// TwinCAT 3 PLC project Field_IO
// ProgramVersion: 3.1.4023.0
// libraries:
//   Tc2_Standard, * (Beckhoff Automation GmbH)
//   Tc2_System, * (Beckhoff Automation GmbH)
//   Tc3_Module, * (Beckhoff Automation GmbH)
// project tree:
//   / PlcTask.TcTTO
//   POUs/ Flasher.TcPOU, HB_M2S.TcPOU, MAIN.TcPOU, HB_S2M.TcPOU
// real-time tasks:
//   TASK IO: cycle T#1ms, priority 1, ADS port 301
//   TASK EIP_Sync_Task: cycle T#2ms, priority 2, ADS port 302
//   TASK PlcTask: cycle T#3ms, priority 3, ADS port 350
// I/O:
//   DEVICE Field_Network (TC3 EIP Adapter), AmsNetId 0.0.0.0.3.1
//     BFIO (TC EtherNet/IP Slave)
//     BSIO (TC EtherNet/IP Slave)
//     Movi_1 (TC EtherNet/IP Slave)
//     Movi_2 (TC EtherNet/IP Slave)
//   DEVICE Device 13 (NOV-DP-RAM)
//   DEVICE SLOT-00 BACKPLANE (EtherCAT), AmsNetId 0.0.0.0.2.1
//     PWR-Supply (EK1200) [EK1200-5000 EtherCAT Power supply (2A E-Bus)]
//       Safety-Ctrl (EL6910) [EL6910, TwinSAFE PLC]
//       License (EL6070-0033) [EL6070-0033 1Ch. Licence key terminal, individual licences]
//       LAS_0600_Slot-01 (EL1018) [EL1018 8Ch. Dig. Input 24V, 10µs]
//       LAS_0600_Slot-02 (EL1018) [EL1018 8Ch. Dig. Input 24V, 10µs]
//       LAS_0600_Slot-03 (EL1018) [EL1018 8Ch. Dig. Input 24V, 10µs]
//       LAS_0600_Slot-04 (EL1904) [EL1904, 4 Ch. Safety Input 24V, TwinSAFE]
//         modules: Module 1 (FSOES)
//       LAS_0600_Slot-05 (EL2008) [EL2008 8Ch. Dig. Output 24V, 0.5A]
//       ECAT-Extension (EK1110) [EK1110 EtherCAT extension]
//     MCP-IOLINK (EP6224-2022) [EP6224-2022 (IO Link Master)]
//       modules: Module 1 (DeviceState Inputs Device), Module 2 (DeviceState Inputs), Module 3 (empty), Module 4 (IO-Link Slave), Module 5 (empty), Module 6 (empty)
//   DEVICE SLOT-01-X600-X601 (EtherCAT) (disabled), AmsNetId 0.0.0.0.4.1
//   DEVICE SLOT-02-X600-X601 (EtherCAT), AmsNetId 0.0.0.0.5.1
//   DEVICE SLOT-03-X600-X601 (EtherCAT), AmsNetId 0.0.0.0.7.1
//     BSIO_LLUB-0635_1 (EP1957-0022) [EP1957, 8Ch. Safety Input 24V, 4Ch. Safety Output 24V, 0.5A, TwinSAFE]
//       modules: Module 1 (FSOE), Module 2 (FSOUT), Module 3 (DEVICEIO), Module 4 (FSLOGIC)
//     BFIO_LLUB-0635_1 (EP2338-0002) [EP2338-0002 8 Ch. Dig. Input/Output 24V, 0,5A, M12]
//     BSIO_LLUB-0636_1 (EP1957-0022) [EP1957, 8Ch. Safety Input 24V, 4Ch. Safety Output 24V, 0.5A, TwinSAFE]
//       modules: Module 1 (FSOE), Module 2 (FSOUT), Module 3 (DEVICEIO), Module 4 (FSLOGIC)
//     BFIO_LLUB-0636_1(EP2338-0002) [EP2338-0002 8 Ch. Dig. Input/Output 24V, 0,5A, M12]
//     MOVI_LLUB-0637 (MOVIMOT+MFE72A) [MOVIMOT+MFE72A]
//     LLU-0200 Coupler (EK1100) [EK1100 EtherCAT Coupler (2A E-Bus)]
//       LLU_0200_Slot-01 (EL1018) [EL1018 8Ch. Dig. Input 24V, 10µs]
//       LLU_0200_Slot-02(EL1018) [EL1018 8Ch. Dig. Input 24V, 10µs]
//       LLU_0200_Slot-03 (EL1018) [EL1018 8Ch. Dig. Input 24V, 10µs]
//       LLU_0200_Slot-04 (EL1904) [EL1904, 4 Ch. Safety Input 24V, TwinSAFE]
//         modules: Module 1 (FSOES)
//       LLU_0200_Slot-05 (EL2008) [EL2008 8Ch. Dig. Output 24V, 0.5A]
//       Slot-06 (EK1110) [EK1110 EtherCAT extension]
//     MOVI_LLUB-0241 (MOVIMOT+MFE72A) [MOVIMOT+MFE72A]
//     MOVI_LLUB-0251 (MOVIMOT+MFE72A) [MOVIMOT+MFE72A]
//     BSIO_LLUB-0639_1  (EP1957-0022) [EP1957, 8Ch. Safety Input 24V, 4Ch. Safety Output 24V, 0.5A, TwinSAFE]
//       modules: Module 1 (FSOE), Module 2 (FSOUT), Module 3 (DEVICEIO), Module 4 (FSLOGIC)
//     IOLINK_LLUB-0639_1 (EP6224-2022) [EP6224-2022 (IO Link Master)]
//       modules: Module 1 (DeviceState Inputs Device), Module 2 (DeviceState Inputs), Module 3 (empty), Module 4 (IO-Link Slave), Module 5 (empty), Module 6 (empty)
//     MOVI_LLUB-0639 (MOVITRAC+FSE24B) [MOVITRAC+FSE24B]
//     BSIO_LLUB-0639_2 (EP1957-0022) [EP1957, 8Ch. Safety Input 24V, 4Ch. Safety Output 24V, 0.5A, TwinSAFE]
//       modules: Module 1 (FSOE), Module 2 (FSOUT), Module 3 (DEVICEIO), Module 4 (FSLOGIC)
//     BSIO_LLUB-0639_2 (EP2338-0002) [EP2338-0002 8 Ch. Dig. Input/Output 24V, 0,5A, M12]
//     BSIO_LLUB-0639_3 (EP1957-0022) [EP1957, 8Ch. Safety Input 24V, 4Ch. Safety Output 24V, 0.5A, TwinSAFE]
//       modules: Module 1 (FSOE), Module 2 (FSOUT), Module 3 (DEVICEIO), Module 4 (FSLOGIC)
//     MOVI_LLUB-0638 (MOVIMOT+MFE72A) [MOVIMOT+MFE72A]
//     MOVI_LLUB-0636 (MOVITRAC+FSE24B) [MOVITRAC+FSE24B]
//     MOVI_LLUB-0635 (MOVITRAC+FSE24B) [MOVITRAC+FSE24B]
//   DEVICE SLOT-04-X600-X601 (EtherCAT), AmsNetId 0.0.0.0.8.1
//     BFIO-LASB-0622_1 (EP2338-0002) [EP2338-0002 8 Ch. Dig. Input/Output 24V, 0,5A, M12]
//     MOVI-LASB-0625 (MOVIMOT+MFE72A) [MOVIMOT+MFE72A]
//     MOVI-LASR-0624 (MOVIMOT+MFE72A) [MOVIMOT+MFE72A]
//     BFIO-LASB-0620_1 (EP2338-0002) [EP2338-0002 8 Ch. Dig. Input/Output 24V, 0,5A, M12]
//     BSIO-LASB-0622_1 (EP1957-0022) [EP1957, 8Ch. Safety Input 24V, 4Ch. Safety Output 24V, 0.5A, TwinSAFE]
//       modules: Module 1 (FSOE), Module 2 (FSOUT), Module 3 (DEVICEIO), Module 4 (FSLOGIC)
//     MOVI-LASB-0626 (MOVIMOT+MFE72A) [MOVIMOT+MFE72A]
//     MOVI-LASB-0629 (MOVIMOT+MFE72A) [MOVIMOT+MFE72A]
//     MOVI-LASB-0628 (MOVIMOT+MFE72A) [MOVIMOT+MFE72A]
//     MOVI-LASB-0627 (MOVIMOT+MFE72A) [MOVIMOT+MFE72A]
//     BSIO-LASB-0623_1 (EP1957-0022) [EP1957, 8Ch. Safety Input 24V, 4Ch. Safety Output 24V, 0.5A, TwinSAFE]
//       modules: Module 1 (FSOE), Module 2 (FSOUT), Module 3 (DEVICEIO), Module 4 (FSLOGIC)
//     MOVI-LASR-0632 (MOVIMOT+MFE72A) [MOVIMOT+MFE72A]
//     MOVI-LASR-0631 (MOVIMOT+MFE72A) [MOVIMOT+MFE72A]
//     MOVI-LASR-0630 (MOVIMOT+MFE72A) [MOVIMOT+MFE72A]
//     MOVI-LASB-0623 (MOVIMOT+MFE72A) [MOVIMOT+MFE72A]
//     MOVI-LASB-0633 (MOVIMOT+MFE72A) [MOVIMOT+MFE72A]
//     MOVI-LASB-0634 (MOVIMOT+MFE72A) [MOVIMOT+MFE72A]
//     BSIO-LASB-0633_1 (EP1957-0022) [EP1957, 8Ch. Safety Input 24V, 4Ch. Safety Output 24V, 0.5A, TwinSAFE]
//       modules: Module 1 (FSOE), Module 2 (FSOUT), Module 3 (DEVICEIO), Module 4 (FSLOGIC)
//     BSIO-LASB-0629_1 (EP1957-0022) [EP1957, 8Ch. Safety Input 24V, 4Ch. Safety Output 24V, 0.5A, TwinSAFE]
//       modules: Module 1 (FSOE), Module 2 (FSOUT), Module 3 (DEVICEIO), Module 4 (FSLOGIC)
//     BSIO-LASB-0625_1 (EP1957-0022) [EP1957, 8Ch. Safety Input 24V, 4Ch. Safety Output 24V, 0.5A, TwinSAFE]
//       modules: Module 1 (FSOE), Module 2 (FSOUT), Module 3 (DEVICEIO), Module 4 (FSLOGIC)
// variable links:
//   Field_Network (TC3 EIP Adapter) <-> SLOT-00 BACKPLANE (EtherCAT)/MCP-IOLINK (EP6224-2022)
//     BFIO (TC EtherNet/IP Slave)/Assembly 1 (Input/Output)/Inputs/M2S_BFIO_301 <-> Module 4 (IO-Link Slave)/IO-Link Port2_out/Port2: process data[1]
//   Field_Network (TC3 EIP Adapter) <-> SLOT-00 BACKPLANE (EtherCAT)/PWR-Supply (EK1200)/LAS_0600_Slot-01 (EL1018)
//     BFIO (TC EtherNet/IP Slave)/Assembly 1 (Input/Output)/Outputs/S2M_BFIO_1 @bit 4 <-> Channel 5/Input
//   Field_Network (TC3 EIP Adapter) <-> SLOT-00 BACKPLANE (EtherCAT)/PWR-Supply (EK1200)/LAS_0600_Slot-02 (EL1018)
//     BFIO (TC EtherNet/IP Slave)/Assembly 1 (Input/Output)/Outputs/S2M_BFIO_2 @bit 5 <-> Channel 6/Input
//   Field_Network (TC3 EIP Adapter) <-> SLOT-00 BACKPLANE (EtherCAT)/PWR-Supply (EK1200)/LAS_0600_Slot-03 (EL1018)
//     BFIO (TC EtherNet/IP Slave)/Assembly 1 (Input/Output)/Outputs/S2M_BFIO_3 <-> Channel 1/Input
//     BFIO (TC EtherNet/IP Slave)/Assembly 1 (Input/Output)/Outputs/S2M_BFIO_3 @bit {1..7} <-> Channel {2..8}/Input  (7 links)
//   Field_Network (TC3 EIP Adapter) <-> SLOT-00 BACKPLANE (EtherCAT)/PWR-Supply (EK1200)/LAS_0600_Slot-04 (EL1904)
//     BSIO (TC EtherNet/IP Slave)/Assembly 3 (Input/Output)/Outputs/S2M_BSIO__11 @bit 3 <-> Module 1 (FSOES)/TxPDO/FSOE/InputChannel4
//   Field_Network (TC3 EIP Adapter) <-> SLOT-00 BACKPLANE (EtherCAT)/PWR-Supply (EK1200)/LAS_0600_Slot-05 (EL2008)
//     BFIO (TC EtherNet/IP Slave)/Assembly 1 (Input/Output)/Inputs/M2S_BFIO_1 <-> Channel 1/Output
//     BFIO (TC EtherNet/IP Slave)/Assembly 1 (Input/Output)/Inputs/M2S_BFIO_1 @bit 1 <-> Channel 2/Output
//     BFIO (TC EtherNet/IP Slave)/Assembly 1 (Input/Output)/Inputs/M2S_BFIO_1 @bit 4 <-> Channel 5/Output
//     BFIO (TC EtherNet/IP Slave)/Assembly 1 (Input/Output)/Inputs/M2S_BFIO_1 @bit 5 <-> Channel 6/Output
//     BFIO (TC EtherNet/IP Slave)/Assembly 1 (Input/Output)/Inputs/M2S_BFIO_1 @bit 6 <-> Channel 7/Output
//   Field_Network (TC3 EIP Adapter) <-> SLOT-00 BACKPLANE (EtherCAT)/PWR-Supply (EK1200)/Safety-Ctrl (EL6910)
//     BSIO (TC EtherNet/IP Slave)/Assembly 3 (Input/Output)/Outputs/S2M_BSIO_2 @bit 1 <-> StandardInputs/Standard Out Var 27
//     BSIO (TC EtherNet/IP Slave)/Assembly 3 (Input/Output)/Outputs/S2M_BSIO_2 @bit 2 <-> StandardInputs/Standard Out Var 30
//     BSIO (TC EtherNet/IP Slave)/Assembly 3 (Input/Output)/Outputs/S2M_BSIO_2 @bit 3 <-> StandardInputs/Standard Out Var 31
//     BSIO (TC EtherNet/IP Slave)/Assembly 3 (Input/Output)/Outputs/S2M_BSIO_2 @bit 4 <-> StandardInputs/Standard Out Var 32
//     BSIO (TC EtherNet/IP Slave)/Assembly 3 (Input/Output)/Outputs/S2M_BSIO_2 @bit 5 <-> StandardInputs/Standard Out Var 33
//     BSIO (TC EtherNet/IP Slave)/Assembly 3 (Input/Output)/Outputs/S2M_BSIO_2 @bit 6 <-> StandardInputs/Standard Out Var 34
//     BSIO (TC EtherNet/IP Slave)/Assembly 3 (Input/Output)/Outputs/S2M_BSIO_2 @bit 7 <-> StandardInputs/Standard Out Var 35
//     BSIO (TC EtherNet/IP Slave)/Assembly 3 (Input/Output)/Outputs/S2M_BSIO_2 <-> StandardInputs/Standard Out Var 37
//   Field_Network (TC3 EIP Adapter) <-> SLOT-03-X600-X601 (EtherCAT)/BFIO_LLUB-0635_1 (EP2338-0002)
//     BFIO (TC EtherNet/IP Slave)/Assembly 1 (Input/Output)/Inputs/M2S_BFIO_11 @bit 1 <-> Channel 10/Output
//     BFIO (TC EtherNet/IP Slave)/Assembly 1 (Input/Output)/Inputs/M2S_BFIO_11 @bit 2 <-> Channel 11/Output
//     BFIO (TC EtherNet/IP Slave)/Assembly 1 (Input/Output)/Inputs/M2S_BFIO_11 @bit 3 <-> Channel 12/Output
//     BFIO (TC EtherNet/IP Slave)/Assembly 1 (Input/Output)/Inputs/M2S_BFIO_11 @bit 4 <-> Channel 13/Output
//     BFIO (TC EtherNet/IP Slave)/Assembly 1 (Input/Output)/Inputs/M2S_BFIO_11 @bit 6 <-> Channel 15/Output
//     BFIO (TC EtherNet/IP Slave)/Assembly 1 (Input/Output)/Inputs/M2S_BFIO_11 @bit 7 <-> Channel 16/Output
//   Field_Network (TC3 EIP Adapter) <-> SLOT-03-X600-X601 (EtherCAT)/BFIO_LLUB-0636_1(EP2338-0002)
//     BFIO (TC EtherNet/IP Slave)/Assembly 1 (Input/Output)/Inputs/M2S_BFIO_12 @bit 1 <-> Channel 10/Output
//     BFIO (TC EtherNet/IP Slave)/Assembly 1 (Input/Output)/Inputs/M2S_BFIO_12 @bit 4 <-> Channel 13/Output
//     BFIO (TC EtherNet/IP Slave)/Assembly 1 (Input/Output)/Inputs/M2S_BFIO_12 @bit 5 <-> Channel 14/Output
//     BFIO (TC EtherNet/IP Slave)/Assembly 1 (Input/Output)/Inputs/M2S_BFIO_12 @bit 6 <-> Channel 15/Output
//     BFIO (TC EtherNet/IP Slave)/Assembly 1 (Input/Output)/Inputs/M2S_BFIO_12 <-> Channel 9/Output
//     BFIO (TC EtherNet/IP Slave)/Assembly 1 (Input/Output)/Outputs/S2M_BFIO_14 @bit 1 <-> Channel 2/Input
//     BFIO (TC EtherNet/IP Slave)/Assembly 1 (Input/Output)/Outputs/S2M_BFIO_14 @bit 2 <-> Channel 3/Input
//     BFIO (TC EtherNet/IP Slave)/Assembly 1 (Input/Output)/Outputs/S2M_BFIO_14 @bit 3 <-> Channel 4/Input
//     BFIO (TC EtherNet/IP Slave)/Assembly 1 (Input/Output)/Outputs/S2M_BFIO_14 @bit 4 <-> Channel 5/Input
//     BFIO (TC EtherNet/IP Slave)/Assembly 1 (Input/Output)/Outputs/S2M_BFIO_14 @bit 6 <-> Channel 7/Input
//     BFIO (TC EtherNet/IP Slave)/Assembly 1 (Input/Output)/Outputs/S2M_BFIO_14 @bit 7 <-> Channel 8/Input
//   Field_Network (TC3 EIP Adapter) <-> SLOT-03-X600-X601 (EtherCAT)/BSIO_LLUB-0635_1 (EP1957-0022)
//     BSIO (TC EtherNet/IP Slave)/Assembly 3 (Input/Output)/Outputs/S2M_BSIO__33 @bit 7 <-> Module 1 (FSOE)/FSoE Inputs/FSOE/FSIN Module 4.Channel 2.Input
//   Field_Network (TC3 EIP Adapter) <-> SLOT-03-X600-X601 (EtherCAT)/BSIO_LLUB-0636_1 (EP1957-0022)
//     BSIO (TC EtherNet/IP Slave)/Assembly 3 (Input/Output)/Outputs/S2M_BSIO__34 @bit 1 <-> Module 1 (FSOE)/FSoE Inputs/FSOE/FSIN Module 1.Channel 2.Input
//     BSIO (TC EtherNet/IP Slave)/Assembly 3 (Input/Output)/Outputs/S2M_BSIO__34 @bit 2 <-> Module 1 (FSOE)/FSoE Inputs/FSOE/FSIN Module 2.Channel 1.Input
//     BSIO (TC EtherNet/IP Slave)/Assembly 3 (Input/Output)/Outputs/S2M_BSIO__34 @bit 3 <-> Module 1 (FSOE)/FSoE Inputs/FSOE/FSIN Module 2.Channel 2.Input
//     BSIO (TC EtherNet/IP Slave)/Assembly 3 (Input/Output)/Outputs/S2M_BSIO__34 @bit 4 <-> Module 1 (FSOE)/FSoE Inputs/FSOE/FSIN Module 3.Channel 1.Input
//     BSIO (TC EtherNet/IP Slave)/Assembly 3 (Input/Output)/Outputs/S2M_BSIO__34 @bit 5 <-> Module 1 (FSOE)/FSoE Inputs/FSOE/FSIN Module 3.Channel 2.Input
//     BSIO (TC EtherNet/IP Slave)/Assembly 3 (Input/Output)/Outputs/S2M_BSIO__34 @bit 6 <-> Module 1 (FSOE)/FSoE Inputs/FSOE/FSIN Module 4.Channel 1.Input
//     BSIO (TC EtherNet/IP Slave)/Assembly 3 (Input/Output)/Outputs/S2M_BSIO__34 @bit 7 <-> Module 1 (FSOE)/FSoE Inputs/FSOE/FSIN Module 4.Channel 2.Input
//   Field_Network (TC3 EIP Adapter) <-> SLOT-03-X600-X601 (EtherCAT)/BSIO_LLUB-0639_1  (EP1957-0022)
//     BSIO (TC EtherNet/IP Slave)/Assembly 3 (Input/Output)/Outputs/S2M_BSIO__35 @bit 1 <-> Module 1 (FSOE)/FSoE Inputs/FSOE/FSIN Module 1.Channel 2.Input
//     BSIO (TC EtherNet/IP Slave)/Assembly 3 (Input/Output)/Outputs/S2M_BSIO__35 @bit 2 <-> Module 1 (FSOE)/FSoE Inputs/FSOE/FSIN Module 2.Channel 1.Input
//     BSIO (TC EtherNet/IP Slave)/Assembly 3 (Input/Output)/Outputs/S2M_BSIO__35 @bit 4 <-> Module 1 (FSOE)/FSoE Inputs/FSOE/FSIN Module 3.Channel 1.Input
//     BSIO (TC EtherNet/IP Slave)/Assembly 3 (Input/Output)/Outputs/S2M_BSIO__35 @bit 5 <-> Module 1 (FSOE)/FSoE Inputs/FSOE/FSIN Module 3.Channel 2.Input
//   Field_Network (TC3 EIP Adapter) <-> SLOT-03-X600-X601 (EtherCAT)/BSIO_LLUB-0639_2 (EP1957-0022)
//     BSIO (TC EtherNet/IP Slave)/Assembly 3 (Input/Output)/Outputs/S2M_BSIO__36 @bit 2 <-> Module 1 (FSOE)/FSoE Inputs/FSOE/FSIN Module 2.Channel 1.Input
//     BSIO (TC EtherNet/IP Slave)/Assembly 3 (Input/Output)/Outputs/S2M_BSIO__36 @bit 3 <-> Module 1 (FSOE)/FSoE Inputs/FSOE/FSIN Module 2.Channel 2.Input
//     BSIO (TC EtherNet/IP Slave)/Assembly 3 (Input/Output)/Outputs/S2M_BSIO__36 @bit 6 <-> Module 1 (FSOE)/FSoE Inputs/FSOE/FSIN Module 4.Channel 1.Input
//     BSIO (TC EtherNet/IP Slave)/Assembly 3 (Input/Output)/Outputs/S2M_BSIO__36 @bit 7 <-> Module 1 (FSOE)/FSoE Inputs/FSOE/FSIN Module 4.Channel 2.Input
//   Field_Network (TC3 EIP Adapter) <-> SLOT-03-X600-X601 (EtherCAT)/BSIO_LLUB-0639_2 (EP2338-0002)
//     BFIO (TC EtherNet/IP Slave)/Assembly 1 (Input/Output)/Inputs/M2S_BFIO_13 @bit 1 <-> Channel 10/Output
//     BFIO (TC EtherNet/IP Slave)/Assembly 1 (Input/Output)/Inputs/M2S_BFIO_13 @bit 5 <-> Channel 14/Output
//     BFIO (TC EtherNet/IP Slave)/Assembly 1 (Input/Output)/Inputs/M2S_BFIO_13 @bit 6 <-> Channel 15/Output
//     BFIO (TC EtherNet/IP Slave)/Assembly 1 (Input/Output)/Inputs/M2S_BFIO_13 <-> Channel 9/Output
//     BFIO (TC EtherNet/IP Slave)/Assembly 1 (Input/Output)/Outputs/S2M_BFIO_15 @bit 1 <-> Channel 2/Input
//     BFIO (TC EtherNet/IP Slave)/Assembly 1 (Input/Output)/Outputs/S2M_BFIO_15 @bit 2 <-> Channel 3/Input
//     BFIO (TC EtherNet/IP Slave)/Assembly 1 (Input/Output)/Outputs/S2M_BFIO_15 @bit 3 <-> Channel 4/Input
//     BFIO (TC EtherNet/IP Slave)/Assembly 1 (Input/Output)/Outputs/S2M_BFIO_15 @bit 4 <-> Channel 5/Input
//     BFIO (TC EtherNet/IP Slave)/Assembly 1 (Input/Output)/Outputs/S2M_BFIO_15 @bit 7 <-> Channel 8/Input
//   Field_Network (TC3 EIP Adapter) <-> SLOT-03-X600-X601 (EtherCAT)/BSIO_LLUB-0639_3 (EP1957-0022)
//     BSIO (TC EtherNet/IP Slave)/Assembly 3 (Input/Output)/Outputs/S2M_BSIO__37 <-> Module 1 (FSOE)/FSoE Inputs/FSOE/FSIN Module 1.Channel 1.Input
//     BSIO (TC EtherNet/IP Slave)/Assembly 3 (Input/Output)/Outputs/S2M_BSIO__37 @bit 3 <-> Module 1 (FSOE)/FSoE Inputs/FSOE/FSIN Module 2.Channel 2.Input
//     BSIO (TC EtherNet/IP Slave)/Assembly 3 (Input/Output)/Outputs/S2M_BSIO__37 @bit 7 <-> Module 1 (FSOE)/FSoE Inputs/FSOE/FSIN Module 4.Channel 2.Input
//   Field_Network (TC3 EIP Adapter) <-> SLOT-03-X600-X601 (EtherCAT)/IOLINK_LLUB-0639_1 (EP6224-2022)
//     BFIO (TC EtherNet/IP Slave)/Assembly 1 (Input/Output)/Inputs/M2S_BFIO_301 <-> Module 4 (IO-Link Slave)/IO-Link Port2_out/Port2: process data[1]
//     BFIO (TC EtherNet/IP Slave)/Assembly 1 (Input/Output)/Inputs/M2S_BFIO_302 <-> Module 4 (IO-Link Slave)/IO-Link Port2_out/Port2: process data[2]
//     BFIO (TC EtherNet/IP Slave)/Assembly 1 (Input/Output)/Inputs/M2S_BFIO_307 <-> Module 4 (IO-Link Slave)/IO-Link Port2_out/Port2: process data[7]
//   Field_Network (TC3 EIP Adapter) <-> SLOT-03-X600-X601 (EtherCAT)/LLU-0200 Coupler (EK1100)/LLU_0200_Slot-01 (EL1018)
//     BFIO (TC EtherNet/IP Slave)/Assembly 1 (Input/Output)/Outputs/S2M_BFIO_10 <-> Channel 1/Input
//     BFIO (TC EtherNet/IP Slave)/Assembly 1 (Input/Output)/Outputs/S2M_BFIO_10 @bit 1 <-> Channel 2/Input
//     BFIO (TC EtherNet/IP Slave)/Assembly 1 (Input/Output)/Outputs/S2M_BFIO_10 @bit 4 <-> Channel 5/Input
//     BFIO (TC EtherNet/IP Slave)/Assembly 1 (Input/Output)/Outputs/S2M_BFIO_10 @bit 5 <-> Channel 6/Input
//     BFIO (TC EtherNet/IP Slave)/Assembly 1 (Input/Output)/Outputs/S2M_BFIO_10 @bit 6 <-> Channel 7/Input
//   Field_Network (TC3 EIP Adapter) <-> SLOT-03-X600-X601 (EtherCAT)/LLU-0200 Coupler (EK1100)/LLU_0200_Slot-02(EL1018)
//     BFIO (TC EtherNet/IP Slave)/Assembly 1 (Input/Output)/Outputs/S2M_BFIO_11 @bit 1 <-> Channel 2/Input
//     BFIO (TC EtherNet/IP Slave)/Assembly 1 (Input/Output)/Outputs/S2M_BFIO_11 @bit 2 <-> Channel 3/Input
//     BFIO (TC EtherNet/IP Slave)/Assembly 1 (Input/Output)/Outputs/S2M_BFIO_11 @bit 6 <-> Channel 7/Input
//     BFIO (TC EtherNet/IP Slave)/Assembly 1 (Input/Output)/Outputs/S2M_BFIO_11 @bit 7 <-> Channel 8/Input
//   Field_Network (TC3 EIP Adapter) <-> SLOT-03-X600-X601 (EtherCAT)/LLU-0200 Coupler (EK1100)/LLU_0200_Slot-03 (EL1018)
//     BFIO (TC EtherNet/IP Slave)/Assembly 1 (Input/Output)/Outputs/S2M_BFIO_12 @bit 4 <-> Channel 5/Input
//   Field_Network (TC3 EIP Adapter) <-> SLOT-03-X600-X601 (EtherCAT)/LLU-0200 Coupler (EK1100)/LLU_0200_Slot-04 (EL1904)
//     BSIO (TC EtherNet/IP Slave)/Assembly 3 (Input/Output)/Outputs/S2M_BSIO__31 @bit 3 <-> Module 1 (FSOES)/TxPDO/FSOE/InputChannel4
//   Field_Network (TC3 EIP Adapter) <-> SLOT-03-X600-X601 (EtherCAT)/LLU-0200 Coupler (EK1100)/LLU_0200_Slot-05 (EL2008)
//     BFIO (TC EtherNet/IP Slave)/Assembly 1 (Input/Output)/Inputs/M2S_BFIO_10 @bit {1..7} <-> Channel {2..8}/Output  (7 links)
//   Field_Network (TC3 EIP Adapter) <-> SLOT-03-X600-X601 (EtherCAT)/MOVI_LLUB-0241 (MOVIMOT+MFE72A)
//     Movi_1 (TC EtherNet/IP Slave)/Assembly 2 (Input/Output)/Inputs/Movi_14 <-> OutputData1 (Standard 10 PO)/PO 0001
//     Movi_1 (TC EtherNet/IP Slave)/Assembly 2 (Input/Output)/Inputs/Movi_14 @bit 32 <-> OutputData1 (Standard 10 PO)/PO 0003
//     Movi_1 (TC EtherNet/IP Slave)/Assembly 2 (Input/Output)/Inputs/Movi_14 @bit 48 <-> OutputData1 (Standard 10 PO)/PO 0004
//     Movi_1 (TC EtherNet/IP Slave)/Assembly 2 (Input/Output)/Inputs/Movi_14 @bit 64 <-> OutputData1 (Standard 10 PO)/PO 0005
//     Movi_1 (TC EtherNet/IP Slave)/Assembly 2 (Input/Output)/Inputs/Movi_14 @bit 80 <-> OutputData1 (Standard 10 PO)/PO 0006
//     Movi_1 (TC EtherNet/IP Slave)/Assembly 2 (Input/Output)/Inputs/Movi_14 @bit 112 <-> OutputData1 (Standard 10 PO)/PO 0008
//     Movi_1 (TC EtherNet/IP Slave)/Assembly 2 (Input/Output)/Inputs/Movi_14 @bit 128 <-> OutputData1 (Standard 10 PO)/PO 0009
//     Movi_1 (TC EtherNet/IP Slave)/Assembly 2 (Input/Output)/Inputs/Movi_14 @bit 144 <-> OutputData1 (Standard 10 PO)/PO 0010
//   Field_Network (TC3 EIP Adapter) <-> SLOT-03-X600-X601 (EtherCAT)/MOVI_LLUB-0251 (MOVIMOT+MFE72A)
//     Movi_1 (TC EtherNet/IP Slave)/Assembly 2 (Input/Output)/Inputs/Movi_15 <-> OutputData1 (Standard 10 PO)/PO 0001
//     Movi_1 (TC EtherNet/IP Slave)/Assembly 2 (Input/Output)/Inputs/Movi_15 @bit 16 <-> OutputData1 (Standard 10 PO)/PO 0002
//     Movi_1 (TC EtherNet/IP Slave)/Assembly 2 (Input/Output)/Inputs/Movi_15 @bit 32 <-> OutputData1 (Standard 10 PO)/PO 0003
//     Movi_1 (TC EtherNet/IP Slave)/Assembly 2 (Input/Output)/Inputs/Movi_15 @bit 64 <-> OutputData1 (Standard 10 PO)/PO 0005
//     Movi_1 (TC EtherNet/IP Slave)/Assembly 2 (Input/Output)/Inputs/Movi_15 @bit 80 <-> OutputData1 (Standard 10 PO)/PO 0006
//     Movi_1 (TC EtherNet/IP Slave)/Assembly 2 (Input/Output)/Inputs/Movi_15 @bit 96 <-> OutputData1 (Standard 10 PO)/PO 0007
//     Movi_1 (TC EtherNet/IP Slave)/Assembly 2 (Input/Output)/Inputs/Movi_15 @bit 112 <-> OutputData1 (Standard 10 PO)/PO 0008
//   Field_Network (TC3 EIP Adapter) <-> SLOT-03-X600-X601 (EtherCAT)/MOVI_LLUB-0635 (MOVITRAC+FSE24B)
//     Movi_1 (TC EtherNet/IP Slave)/Assembly 2 (Input/Output)/Inputs/Movi_19 <-> OutputData1  (Standard 3 PO)/PO 0001
//     Movi_1 (TC EtherNet/IP Slave)/Assembly 2 (Input/Output)/Inputs/Movi_19 @bit 2 <-> OutputData1  (Standard 3 PO)/PO 0003
//   Field_Network (TC3 EIP Adapter) <-> SLOT-03-X600-X601 (EtherCAT)/MOVI_LLUB-0636 (MOVITRAC+FSE24B)
//     Movi_1 (TC EtherNet/IP Slave)/Assembly 2 (Input/Output)/Inputs/Movi_18 <-> OutputData1  (Standard 3 PO)/PO 0001
//   Field_Network (TC3 EIP Adapter) <-> SLOT-03-X600-X601 (EtherCAT)/MOVI_LLUB-0638 (MOVIMOT+MFE72A)
//     Movi_1 (TC EtherNet/IP Slave)/Assembly 2 (Input/Output)/Inputs/Movi_17 <-> OutputData1 (Standard 10 PO)/PO 0001
//     Movi_1 (TC EtherNet/IP Slave)/Assembly 2 (Input/Output)/Inputs/Movi_17 @bit 16 <-> OutputData1 (Standard 10 PO)/PO 0002
//     Movi_1 (TC EtherNet/IP Slave)/Assembly 2 (Input/Output)/Inputs/Movi_17 @bit 80 <-> OutputData1 (Standard 10 PO)/PO 0006
//     Movi_1 (TC EtherNet/IP Slave)/Assembly 2 (Input/Output)/Inputs/Movi_17 @bit 96 <-> OutputData1 (Standard 10 PO)/PO 0007
//     Movi_1 (TC EtherNet/IP Slave)/Assembly 2 (Input/Output)/Inputs/Movi_17 @bit 112 <-> OutputData1 (Standard 10 PO)/PO 0008
//   Field_Network (TC3 EIP Adapter) <-> SLOT-03-X600-X601 (EtherCAT)/MOVI_LLUB-0639 (MOVITRAC+FSE24B)
//     Movi_1 (TC EtherNet/IP Slave)/Assembly 2 (Input/Output)/Inputs/Movi_16 <-> OutputData1  (Standard 3 PO)/PO 0001
//     Movi_1 (TC EtherNet/IP Slave)/Assembly 2 (Input/Output)/Inputs/Movi_16 @bit 16 <-> OutputData1  (Standard 3 PO)/PO 0002
//     Movi_1 (TC EtherNet/IP Slave)/Assembly 2 (Input/Output)/Inputs/Movi_16 @bit 32 <-> OutputData1  (Standard 3 PO)/PO 0003
//   Field_Network (TC3 EIP Adapter) <-> SLOT-04-X600-X601 (EtherCAT)/BFIO-LASB-0620_1 (EP2338-0002)
//     BFIO (TC EtherNet/IP Slave)/Assembly 1 (Input/Output)/Inputs/M2S_BFIO_3 @bit 5 <-> Channel 14/Output
//     BFIO (TC EtherNet/IP Slave)/Assembly 1 (Input/Output)/Inputs/M2S_BFIO_3 <-> Channel 9/Output
//     BFIO (TC EtherNet/IP Slave)/Assembly 1 (Input/Output)/Outputs/S2M_BFIO_5 @bit 2 <-> Channel 3/Input
//     BFIO (TC EtherNet/IP Slave)/Assembly 1 (Input/Output)/Outputs/S2M_BFIO_5 @bit 3 <-> Channel 4/Input
//     BFIO (TC EtherNet/IP Slave)/Assembly 1 (Input/Output)/Outputs/S2M_BFIO_5 @bit 4 <-> Channel 5/Input
//   Field_Network (TC3 EIP Adapter) <-> SLOT-04-X600-X601 (EtherCAT)/BFIO-LASB-0622_1 (EP2338-0002)
//     BFIO (TC EtherNet/IP Slave)/Assembly 1 (Input/Output)/Inputs/M2S_BFIO_2 @bit 3 <-> Channel 12/Output
//     BFIO (TC EtherNet/IP Slave)/Assembly 1 (Input/Output)/Inputs/M2S_BFIO_2 @bit 4 <-> Channel 13/Output
//     BFIO (TC EtherNet/IP Slave)/Assembly 1 (Input/Output)/Inputs/M2S_BFIO_2 @bit 5 <-> Channel 14/Output
//     BFIO (TC EtherNet/IP Slave)/Assembly 1 (Input/Output)/Inputs/M2S_BFIO_2 <-> Channel 9/Output
//     BFIO (TC EtherNet/IP Slave)/Assembly 1 (Input/Output)/Outputs/S2M_BFIO_4 @bit 1 <-> Channel 2/Input
//     BFIO (TC EtherNet/IP Slave)/Assembly 1 (Input/Output)/Outputs/S2M_BFIO_4 @bit 2 <-> Channel 3/Input
//     BFIO (TC EtherNet/IP Slave)/Assembly 1 (Input/Output)/Outputs/S2M_BFIO_4 @bit 3 <-> Channel 4/Input
//     BFIO (TC EtherNet/IP Slave)/Assembly 1 (Input/Output)/Outputs/S2M_BFIO_4 @bit 4 <-> Channel 5/Input
//     BFIO (TC EtherNet/IP Slave)/Assembly 1 (Input/Output)/Outputs/S2M_BFIO_4 @bit 6 <-> Channel 7/Input
//     BFIO (TC EtherNet/IP Slave)/Assembly 1 (Input/Output)/Outputs/S2M_BFIO_4 @bit 7 <-> Channel 8/Input
//   Field_Network (TC3 EIP Adapter) <-> SLOT-04-X600-X601 (EtherCAT)/BSIO-LASB-0622_1 (EP1957-0022)
//     BSIO (TC EtherNet/IP Slave)/Assembly 3 (Input/Output)/Outputs/S2M_BSIO__13 <-> Module 1 (FSOE)/FSoE Inputs/FSOE/FSIN Module 1.Channel 1.Input
//     BSIO (TC EtherNet/IP Slave)/Assembly 3 (Input/Output)/Outputs/S2M_BSIO__13 @bit 1 <-> Module 1 (FSOE)/FSoE Inputs/FSOE/FSIN Module 1.Channel 2.Input
//     BSIO (TC EtherNet/IP Slave)/Assembly 3 (Input/Output)/Outputs/S2M_BSIO__13 @bit 2 <-> Module 1 (FSOE)/FSoE Inputs/FSOE/FSIN Module 2.Channel 1.Input
//     BSIO (TC EtherNet/IP Slave)/Assembly 3 (Input/Output)/Outputs/S2M_BSIO__13 @bit 4 <-> Module 1 (FSOE)/FSoE Inputs/FSOE/FSIN Module 3.Channel 1.Input
//     BSIO (TC EtherNet/IP Slave)/Assembly 3 (Input/Output)/Outputs/S2M_BSIO__13 @bit 5 <-> Module 1 (FSOE)/FSoE Inputs/FSOE/FSIN Module 3.Channel 2.Input
//     BSIO (TC EtherNet/IP Slave)/Assembly 3 (Input/Output)/Outputs/S2M_BSIO__13 @bit 7 <-> Module 1 (FSOE)/FSoE Inputs/FSOE/FSIN Module 4.Channel 2.Input
//   Field_Network (TC3 EIP Adapter) <-> SLOT-04-X600-X601 (EtherCAT)/BSIO-LASB-0623_1 (EP1957-0022)
//     BSIO (TC EtherNet/IP Slave)/Assembly 3 (Input/Output)/Outputs/S2M_BSIO__14 <-> Module 1 (FSOE)/FSoE Inputs/FSOE/FSIN Module 1.Channel 1.Input
//     BSIO (TC EtherNet/IP Slave)/Assembly 3 (Input/Output)/Outputs/S2M_BSIO__14 @bit 1 <-> Module 1 (FSOE)/FSoE Inputs/FSOE/FSIN Module 1.Channel 2.Input
//     BSIO (TC EtherNet/IP Slave)/Assembly 3 (Input/Output)/Outputs/S2M_BSIO__14 @bit 2 <-> Module 1 (FSOE)/FSoE Inputs/FSOE/FSIN Module 2.Channel 1.Input
//     BSIO (TC EtherNet/IP Slave)/Assembly 3 (Input/Output)/Outputs/S2M_BSIO__14 @bit 3 <-> Module 1 (FSOE)/FSoE Inputs/FSOE/FSIN Module 2.Channel 2.Input
//     BSIO (TC EtherNet/IP Slave)/Assembly 3 (Input/Output)/Outputs/S2M_BSIO__14 @bit 4 <-> Module 1 (FSOE)/FSoE Inputs/FSOE/FSIN Module 3.Channel 1.Input
//     BSIO (TC EtherNet/IP Slave)/Assembly 3 (Input/Output)/Outputs/S2M_BSIO__14 @bit 6 <-> Module 1 (FSOE)/FSoE Inputs/FSOE/FSIN Module 4.Channel 1.Input
//     BSIO (TC EtherNet/IP Slave)/Assembly 3 (Input/Output)/Outputs/S2M_BSIO__14 @bit 7 <-> Module 1 (FSOE)/FSoE Inputs/FSOE/FSIN Module 4.Channel 2.Input
//   Field_Network (TC3 EIP Adapter) <-> SLOT-04-X600-X601 (EtherCAT)/BSIO-LASB-0629_1 (EP1957-0022)
//     BSIO (TC EtherNet/IP Slave)/Assembly 3 (Input/Output)/Outputs/S2M_BSIO__16 <-> Module 1 (FSOE)/FSoE Inputs/FSOE/FSIN Module 1.Channel 1.Input
//     BSIO (TC EtherNet/IP Slave)/Assembly 3 (Input/Output)/Outputs/S2M_BSIO__16 @bit 7 <-> Module 1 (FSOE)/FSoE Inputs/FSOE/FSIN Module 4.Channel 2.Input
//   Field_Network (TC3 EIP Adapter) <-> SLOT-04-X600-X601 (EtherCAT)/BSIO-LASB-0633_1 (EP1957-0022)
//     BSIO (TC EtherNet/IP Slave)/Assembly 3 (Input/Output)/Outputs/S2M_BSIO__15 @bit 2 <-> Module 1 (FSOE)/FSoE Inputs/FSOE/FSIN Module 2.Channel 1.Input
//     BSIO (TC EtherNet/IP Slave)/Assembly 3 (Input/Output)/Outputs/S2M_BSIO__15 @bit 3 <-> Module 1 (FSOE)/FSoE Inputs/FSOE/FSIN Module 2.Channel 2.Input
//     BSIO (TC EtherNet/IP Slave)/Assembly 3 (Input/Output)/Outputs/S2M_BSIO__15 @bit 6 <-> Module 1 (FSOE)/FSoE Inputs/FSOE/FSIN Module 4.Channel 1.Input
//     BSIO (TC EtherNet/IP Slave)/Assembly 3 (Input/Output)/Outputs/S2M_BSIO__15 @bit 7 <-> Module 1 (FSOE)/FSoE Inputs/FSOE/FSIN Module 4.Channel 2.Input
//   Field_Network (TC3 EIP Adapter) <-> SLOT-04-X600-X601 (EtherCAT)/MOVI-LASB-0623 (MOVIMOT+MFE72A)
//     Movi_1 (TC EtherNet/IP Slave)/Assembly 2 (Input/Output)/Inputs/Movi_10 <-> OutputData1 (Standard 10 PO)/PO 0001
//     Movi_1 (TC EtherNet/IP Slave)/Assembly 2 (Input/Output)/Inputs/Movi_10 @bit 16 <-> OutputData1 (Standard 10 PO)/PO 0002
//     Movi_1 (TC EtherNet/IP Slave)/Assembly 2 (Input/Output)/Inputs/Movi_10 @bit 80 <-> OutputData1 (Standard 10 PO)/PO 0006
//     Movi_1 (TC EtherNet/IP Slave)/Assembly 2 (Input/Output)/Inputs/Movi_10 @bit 96 <-> OutputData1 (Standard 10 PO)/PO 0007
//     Movi_1 (TC EtherNet/IP Slave)/Assembly 2 (Input/Output)/Outputs/Movi_10 <-> InputData1 (Standard 10 PI)/PI 0001
//     Movi_1 (TC EtherNet/IP Slave)/Assembly 2 (Input/Output)/Outputs/Movi_10 @bit 80 <-> InputData1 (Standard 10 PI)/PI 0006
//   Field_Network (TC3 EIP Adapter) <-> SLOT-04-X600-X601 (EtherCAT)/MOVI-LASB-0625 (MOVIMOT+MFE72A)
//     Movi_1 (TC EtherNet/IP Slave)/Assembly 2 (Input/Output)/Inputs/Movi_1 <-> OutputData1 (Standard 10 PO)/PO 0001
//     Movi_1 (TC EtherNet/IP Slave)/Assembly 2 (Input/Output)/Inputs/Movi_1 @bit 16 <-> OutputData1 (Standard 10 PO)/PO 0002
//     Movi_1 (TC EtherNet/IP Slave)/Assembly 2 (Input/Output)/Inputs/Movi_1 @bit 80 <-> OutputData1 (Standard 10 PO)/PO 0006
//     Movi_1 (TC EtherNet/IP Slave)/Assembly 2 (Input/Output)/Inputs/Movi_1 @bit 96 <-> OutputData1 (Standard 10 PO)/PO 0007
//     Movi_1 (TC EtherNet/IP Slave)/Assembly 2 (Input/Output)/Outputs/Movi_1 <-> InputData1 (Standard 10 PI)/PI 0001
//     Movi_1 (TC EtherNet/IP Slave)/Assembly 2 (Input/Output)/Outputs/Movi_1 @bit 80 <-> InputData1 (Standard 10 PI)/PI 0006
//   Field_Network (TC3 EIP Adapter) <-> SLOT-04-X600-X601 (EtherCAT)/MOVI-LASB-0626 (MOVIMOT+MFE72A)
//     Movi_1 (TC EtherNet/IP Slave)/Assembly 2 (Input/Output)/Inputs/Movi_3 <-> OutputData1 (Standard 10 PO)/PO 0001
//     Movi_1 (TC EtherNet/IP Slave)/Assembly 2 (Input/Output)/Inputs/Movi_3 @bit 80 <-> OutputData1 (Standard 10 PO)/PO 0006
//     Movi_1 (TC EtherNet/IP Slave)/Assembly 2 (Input/Output)/Outputs/Movi_3 <-> InputData1 (Standard 10 PI)/PI 0001
//     Movi_1 (TC EtherNet/IP Slave)/Assembly 2 (Input/Output)/Outputs/Movi_3 @bit 16 <-> InputData1 (Standard 10 PI)/PI 0002
//     Movi_1 (TC EtherNet/IP Slave)/Assembly 2 (Input/Output)/Outputs/Movi_3 @bit 32 <-> InputData1 (Standard 10 PI)/PI 0003
//     Movi_1 (TC EtherNet/IP Slave)/Assembly 2 (Input/Output)/Outputs/Movi_3 @bit 48 <-> InputData1 (Standard 10 PI)/PI 0004
//     Movi_1 (TC EtherNet/IP Slave)/Assembly 2 (Input/Output)/Outputs/Movi_3 @bit 64 <-> InputData1 (Standard 10 PI)/PI 0005
//     Movi_1 (TC EtherNet/IP Slave)/Assembly 2 (Input/Output)/Outputs/Movi_3 @bit 80 <-> InputData1 (Standard 10 PI)/PI 0006
//     Movi_1 (TC EtherNet/IP Slave)/Assembly 2 (Input/Output)/Outputs/Movi_3 @bit 96 <-> InputData1 (Standard 10 PI)/PI 0007
//     Movi_1 (TC EtherNet/IP Slave)/Assembly 2 (Input/Output)/Outputs/Movi_3 @bit 112 <-> InputData1 (Standard 10 PI)/PI 0008
//     Movi_1 (TC EtherNet/IP Slave)/Assembly 2 (Input/Output)/Outputs/Movi_3 @bit 128 <-> InputData1 (Standard 10 PI)/PI 0009
//     Movi_1 (TC EtherNet/IP Slave)/Assembly 2 (Input/Output)/Outputs/Movi_3 @bit 144 <-> InputData1 (Standard 10 PI)/PI 0010
//   Field_Network (TC3 EIP Adapter) <-> SLOT-04-X600-X601 (EtherCAT)/MOVI-LASB-0627 (MOVIMOT+MFE72A)
//     Movi_1 (TC EtherNet/IP Slave)/Assembly 2 (Input/Output)/Inputs/Movi_6 <-> OutputData1 (Standard 10 PO)/PO 0001
//     Movi_1 (TC EtherNet/IP Slave)/Assembly 2 (Input/Output)/Inputs/Movi_6 @bit 16 <-> OutputData1 (Standard 10 PO)/PO 0002
//     Movi_1 (TC EtherNet/IP Slave)/Assembly 2 (Input/Output)/Inputs/Movi_6 @bit 32 <-> OutputData1 (Standard 10 PO)/PO 0003
//     Movi_1 (TC EtherNet/IP Slave)/Assembly 2 (Input/Output)/Inputs/Movi_6 @bit 48 <-> OutputData1 (Standard 10 PO)/PO 0004
//     Movi_1 (TC EtherNet/IP Slave)/Assembly 2 (Input/Output)/Inputs/Movi_6 @bit 64 <-> OutputData1 (Standard 10 PO)/PO 0005
//     Movi_1 (TC EtherNet/IP Slave)/Assembly 2 (Input/Output)/Inputs/Movi_6 @bit 80 <-> OutputData1 (Standard 10 PO)/PO 0006
//     Movi_1 (TC EtherNet/IP Slave)/Assembly 2 (Input/Output)/Inputs/Movi_6 @bit 112 <-> OutputData1 (Standard 10 PO)/PO 0008
//     Movi_1 (TC EtherNet/IP Slave)/Assembly 2 (Input/Output)/Inputs/Movi_6 @bit 128 <-> OutputData1 (Standard 10 PO)/PO 0009
//     Movi_1 (TC EtherNet/IP Slave)/Assembly 2 (Input/Output)/Inputs/Movi_6 @bit 144 <-> OutputData1 (Standard 10 PO)/PO 0010
//     Movi_1 (TC EtherNet/IP Slave)/Assembly 2 (Input/Output)/Outputs/Movi_6 @bit 16 <-> InputData1 (Standard 10 PI)/PI 0002
//     Movi_1 (TC EtherNet/IP Slave)/Assembly 2 (Input/Output)/Outputs/Movi_6 @bit 32 <-> InputData1 (Standard 10 PI)/PI 0003
//     Movi_1 (TC EtherNet/IP Slave)/Assembly 2 (Input/Output)/Outputs/Movi_6 @bit 48 <-> InputData1 (Standard 10 PI)/PI 0004
//     Movi_1 (TC EtherNet/IP Slave)/Assembly 2 (Input/Output)/Outputs/Movi_6 @bit 96 <-> InputData1 (Standard 10 PI)/PI 0007
//     Movi_1 (TC EtherNet/IP Slave)/Assembly 2 (Input/Output)/Outputs/Movi_6 @bit 112 <-> InputData1 (Standard 10 PI)/PI 0008
//     Movi_1 (TC EtherNet/IP Slave)/Assembly 2 (Input/Output)/Outputs/Movi_6 @bit 128 <-> InputData1 (Standard 10 PI)/PI 0009
//     Movi_1 (TC EtherNet/IP Slave)/Assembly 2 (Input/Output)/Outputs/Movi_6 @bit 144 <-> InputData1 (Standard 10 PI)/PI 0010
//   Field_Network (TC3 EIP Adapter) <-> SLOT-04-X600-X601 (EtherCAT)/MOVI-LASB-0628 (MOVIMOT+MFE72A)
//     Movi_1 (TC EtherNet/IP Slave)/Assembly 2 (Input/Output)/Inputs/Movi_5 <-> OutputData1 (Standard 10 PO)/PO 0001
//     Movi_1 (TC EtherNet/IP Slave)/Assembly 2 (Input/Output)/Inputs/Movi_5 @bit 16 <-> OutputData1 (Standard 10 PO)/PO 0002
//     Movi_1 (TC EtherNet/IP Slave)/Assembly 2 (Input/Output)/Inputs/Movi_5 @bit 48 <-> OutputData1 (Standard 10 PO)/PO 0004
//     Movi_1 (TC EtherNet/IP Slave)/Assembly 2 (Input/Output)/Inputs/Movi_5 @bit 64 <-> OutputData1 (Standard 10 PO)/PO 0005
//     Movi_1 (TC EtherNet/IP Slave)/Assembly 2 (Input/Output)/Inputs/Movi_5 @bit 80 <-> OutputData1 (Standard 10 PO)/PO 0006
//     Movi_1 (TC EtherNet/IP Slave)/Assembly 2 (Input/Output)/Inputs/Movi_5 @bit 96 <-> OutputData1 (Standard 10 PO)/PO 0007
//     Movi_1 (TC EtherNet/IP Slave)/Assembly 2 (Input/Output)/Inputs/Movi_5 @bit 112 <-> OutputData1 (Standard 10 PO)/PO 0008
//     Movi_1 (TC EtherNet/IP Slave)/Assembly 2 (Input/Output)/Inputs/Movi_5 @bit 128 <-> OutputData1 (Standard 10 PO)/PO 0009
//     Movi_1 (TC EtherNet/IP Slave)/Assembly 2 (Input/Output)/Inputs/Movi_5 @bit 144 <-> OutputData1 (Standard 10 PO)/PO 0010
//     Movi_1 (TC EtherNet/IP Slave)/Assembly 2 (Input/Output)/Outputs/Movi_5 <-> InputData1 (Standard 10 PI)/PI 0001
//     Movi_1 (TC EtherNet/IP Slave)/Assembly 2 (Input/Output)/Outputs/Movi_5 @bit 32 <-> InputData1 (Standard 10 PI)/PI 0003
//     Movi_1 (TC EtherNet/IP Slave)/Assembly 2 (Input/Output)/Outputs/Movi_5 @bit 48 <-> InputData1 (Standard 10 PI)/PI 0004
//     Movi_1 (TC EtherNet/IP Slave)/Assembly 2 (Input/Output)/Outputs/Movi_5 @bit 64 <-> InputData1 (Standard 10 PI)/PI 0005
//     Movi_1 (TC EtherNet/IP Slave)/Assembly 2 (Input/Output)/Outputs/Movi_5 @bit 80 <-> InputData1 (Standard 10 PI)/PI 0006
//     Movi_1 (TC EtherNet/IP Slave)/Assembly 2 (Input/Output)/Outputs/Movi_5 @bit 112 <-> InputData1 (Standard 10 PI)/PI 0008
//     Movi_1 (TC EtherNet/IP Slave)/Assembly 2 (Input/Output)/Outputs/Movi_5 @bit 128 <-> InputData1 (Standard 10 PI)/PI 0009
//     Movi_1 (TC EtherNet/IP Slave)/Assembly 2 (Input/Output)/Outputs/Movi_5 @bit 144 <-> InputData1 (Standard 10 PI)/PI 0010
//   Field_Network (TC3 EIP Adapter) <-> SLOT-04-X600-X601 (EtherCAT)/MOVI-LASB-0629 (MOVIMOT+MFE72A)
//     Movi_1 (TC EtherNet/IP Slave)/Assembly 2 (Input/Output)/Outputs/Movi_4 <-> InputData1 (Standard 10 PI)/PI 0001
//     Movi_1 (TC EtherNet/IP Slave)/Assembly 2 (Input/Output)/Outputs/Movi_4 @bit 16 <-> InputData1 (Standard 10 PI)/PI 0002
//     Movi_1 (TC EtherNet/IP Slave)/Assembly 2 (Input/Output)/Outputs/Movi_4 @bit 32 <-> InputData1 (Standard 10 PI)/PI 0003
//     Movi_1 (TC EtherNet/IP Slave)/Assembly 2 (Input/Output)/Outputs/Movi_4 @bit 48 <-> InputData1 (Standard 10 PI)/PI 0004
//     Movi_1 (TC EtherNet/IP Slave)/Assembly 2 (Input/Output)/Outputs/Movi_4 @bit 64 <-> InputData1 (Standard 10 PI)/PI 0005
//     Movi_1 (TC EtherNet/IP Slave)/Assembly 2 (Input/Output)/Outputs/Movi_4 @bit 80 <-> InputData1 (Standard 10 PI)/PI 0006
//     Movi_1 (TC EtherNet/IP Slave)/Assembly 2 (Input/Output)/Outputs/Movi_4 @bit 96 <-> InputData1 (Standard 10 PI)/PI 0007
//     Movi_1 (TC EtherNet/IP Slave)/Assembly 2 (Input/Output)/Outputs/Movi_4 @bit 112 <-> InputData1 (Standard 10 PI)/PI 0008
//     Movi_1 (TC EtherNet/IP Slave)/Assembly 2 (Input/Output)/Outputs/Movi_4 @bit 144 <-> InputData1 (Standard 10 PI)/PI 0010
//   Field_Network (TC3 EIP Adapter) <-> SLOT-04-X600-X601 (EtherCAT)/MOVI-LASB-0633 (MOVIMOT+MFE72A)
//     Movi_1 (TC EtherNet/IP Slave)/Assembly 2 (Input/Output)/Inputs/Movi_11 @bit 64 <-> OutputData1 (Standard 10 PO)/PO 0005
//     Movi_1 (TC EtherNet/IP Slave)/Assembly 2 (Input/Output)/Inputs/Movi_11 @bit 144 <-> OutputData1 (Standard 10 PO)/PO 0010
//   Field_Network (TC3 EIP Adapter) <-> SLOT-04-X600-X601 (EtherCAT)/MOVI-LASB-0634 (MOVIMOT+MFE72A)
//     Movi_1 (TC EtherNet/IP Slave)/Assembly 2 (Input/Output)/Inputs/Movi_12 @bit 48 <-> OutputData1 (Standard 10 PO)/PO 0004
//     Movi_1 (TC EtherNet/IP Slave)/Assembly 2 (Input/Output)/Inputs/Movi_12 @bit 128 <-> OutputData1 (Standard 10 PO)/PO 0009
//     Movi_1 (TC EtherNet/IP Slave)/Assembly 2 (Input/Output)/Outputs/Movi_12 <-> InputData1 (Standard 10 PI)/PI 0001
//     Movi_1 (TC EtherNet/IP Slave)/Assembly 2 (Input/Output)/Outputs/Movi_12 @bit 16 <-> InputData1 (Standard 10 PI)/PI 0002
//     Movi_1 (TC EtherNet/IP Slave)/Assembly 2 (Input/Output)/Outputs/Movi_12 @bit 48 <-> InputData1 (Standard 10 PI)/PI 0004
//     Movi_1 (TC EtherNet/IP Slave)/Assembly 2 (Input/Output)/Outputs/Movi_12 @bit 64 <-> InputData1 (Standard 10 PI)/PI 0005
//     Movi_1 (TC EtherNet/IP Slave)/Assembly 2 (Input/Output)/Outputs/Movi_12 @bit 80 <-> InputData1 (Standard 10 PI)/PI 0006
//     Movi_1 (TC EtherNet/IP Slave)/Assembly 2 (Input/Output)/Outputs/Movi_12 @bit 96 <-> InputData1 (Standard 10 PI)/PI 0007
//     Movi_1 (TC EtherNet/IP Slave)/Assembly 2 (Input/Output)/Outputs/Movi_12 @bit 112 <-> InputData1 (Standard 10 PI)/PI 0008
//     Movi_1 (TC EtherNet/IP Slave)/Assembly 2 (Input/Output)/Outputs/Movi_12 @bit 128 <-> InputData1 (Standard 10 PI)/PI 0009
//     Movi_1 (TC EtherNet/IP Slave)/Assembly 2 (Input/Output)/Outputs/Movi_12 @bit 144 <-> InputData1 (Standard 10 PI)/PI 0010
//   Field_Network (TC3 EIP Adapter) <-> SLOT-04-X600-X601 (EtherCAT)/MOVI-LASR-0624 (MOVIMOT+MFE72A)
//     Movi_1 (TC EtherNet/IP Slave)/Assembly 2 (Input/Output)/Inputs/Movi_2 @bit 64 <-> OutputData1 (Standard 10 PO)/PO 0005
//     Movi_1 (TC EtherNet/IP Slave)/Assembly 2 (Input/Output)/Inputs/Movi_2 @bit 80 <-> OutputData1 (Standard 10 PO)/PO 0006
//     Movi_1 (TC EtherNet/IP Slave)/Assembly 2 (Input/Output)/Inputs/Movi_2 @bit 144 <-> OutputData1 (Standard 10 PO)/PO 0010
//   Field_Network (TC3 EIP Adapter) <-> SLOT-04-X600-X601 (EtherCAT)/MOVI-LASR-0630 (MOVIMOT+MFE72A)
//     Movi_1 (TC EtherNet/IP Slave)/Assembly 2 (Input/Output)/Inputs/Movi_9 @bit 16 <-> OutputData1 (Standard 10 PO)/PO 0002
//     Movi_1 (TC EtherNet/IP Slave)/Assembly 2 (Input/Output)/Inputs/Movi_9 @bit 32 <-> OutputData1 (Standard 10 PO)/PO 0003
//     Movi_1 (TC EtherNet/IP Slave)/Assembly 2 (Input/Output)/Inputs/Movi_9 @bit 48 <-> OutputData1 (Standard 10 PO)/PO 0004
//     Movi_1 (TC EtherNet/IP Slave)/Assembly 2 (Input/Output)/Inputs/Movi_9 @bit 112 <-> OutputData1 (Standard 10 PO)/PO 0008
//     Movi_1 (TC EtherNet/IP Slave)/Assembly 2 (Input/Output)/Inputs/Movi_9 @bit 128 <-> OutputData1 (Standard 10 PO)/PO 0009
//     Movi_1 (TC EtherNet/IP Slave)/Assembly 2 (Input/Output)/Outputs/Movi_9 @bit 16 <-> InputData1 (Standard 10 PI)/PI 0002
//     Movi_1 (TC EtherNet/IP Slave)/Assembly 2 (Input/Output)/Outputs/Movi_9 @bit 32 <-> InputData1 (Standard 10 PI)/PI 0003
//     Movi_1 (TC EtherNet/IP Slave)/Assembly 2 (Input/Output)/Outputs/Movi_9 @bit 96 <-> InputData1 (Standard 10 PI)/PI 0007
//     Movi_1 (TC EtherNet/IP Slave)/Assembly 2 (Input/Output)/Outputs/Movi_9 @bit 112 <-> InputData1 (Standard 10 PI)/PI 0008
//   Field_Network (TC3 EIP Adapter) <-> SLOT-04-X600-X601 (EtherCAT)/MOVI-LASR-0631 (MOVIMOT+MFE72A)
//     Movi_1 (TC EtherNet/IP Slave)/Assembly 2 (Input/Output)/Inputs/Movi_8 @bit 48 <-> OutputData1 (Standard 10 PO)/PO 0004
//     Movi_1 (TC EtherNet/IP Slave)/Assembly 2 (Input/Output)/Inputs/Movi_8 @bit 64 <-> OutputData1 (Standard 10 PO)/PO 0005
//     Movi_1 (TC EtherNet/IP Slave)/Assembly 2 (Input/Output)/Inputs/Movi_8 @bit 80 <-> OutputData1 (Standard 10 PO)/PO 0006
//     Movi_1 (TC EtherNet/IP Slave)/Assembly 2 (Input/Output)/Inputs/Movi_8 @bit 128 <-> OutputData1 (Standard 10 PO)/PO 0009
//     Movi_1 (TC EtherNet/IP Slave)/Assembly 2 (Input/Output)/Inputs/Movi_8 @bit 144 <-> OutputData1 (Standard 10 PO)/PO 0010
//     Movi_1 (TC EtherNet/IP Slave)/Assembly 2 (Input/Output)/Outputs/Movi_8 @bit 32 <-> InputData1 (Standard 10 PI)/PI 0003
//     Movi_1 (TC EtherNet/IP Slave)/Assembly 2 (Input/Output)/Outputs/Movi_8 @bit 48 <-> InputData1 (Standard 10 PI)/PI 0004
//     Movi_1 (TC EtherNet/IP Slave)/Assembly 2 (Input/Output)/Outputs/Movi_8 @bit 112 <-> InputData1 (Standard 10 PI)/PI 0008
//     Movi_1 (TC EtherNet/IP Slave)/Assembly 2 (Input/Output)/Outputs/Movi_8 @bit 128 <-> InputData1 (Standard 10 PI)/PI 0009
//     Movi_1 (TC EtherNet/IP Slave)/Assembly 2 (Input/Output)/Outputs/Movi_8 @bit 144 <-> InputData1 (Standard 10 PI)/PI 0010
//   Field_Network (TC3 EIP Adapter) <-> SLOT-04-X600-X601 (EtherCAT)/MOVI-LASR-0632 (MOVIMOT+MFE72A)
//     Movi_1 (TC EtherNet/IP Slave)/Assembly 2 (Input/Output)/Inputs/Movi_7 <-> OutputData1 (Standard 10 PO)/PO 0001
//     Movi_1 (TC EtherNet/IP Slave)/Assembly 2 (Input/Output)/Inputs/Movi_7 @bit 16 <-> OutputData1 (Standard 10 PO)/PO 0002
//     Movi_1 (TC EtherNet/IP Slave)/Assembly 2 (Input/Output)/Inputs/Movi_7 @bit 64 <-> OutputData1 (Standard 10 PO)/PO 0005
//     Movi_1 (TC EtherNet/IP Slave)/Assembly 2 (Input/Output)/Inputs/Movi_7 @bit 80 <-> OutputData1 (Standard 10 PO)/PO 0006
//     Movi_1 (TC EtherNet/IP Slave)/Assembly 2 (Input/Output)/Inputs/Movi_7 @bit 96 <-> OutputData1 (Standard 10 PO)/PO 0007
//     Movi_1 (TC EtherNet/IP Slave)/Assembly 2 (Input/Output)/Inputs/Movi_7 @bit 144 <-> OutputData1 (Standard 10 PO)/PO 0010
//     Movi_1 (TC EtherNet/IP Slave)/Assembly 2 (Input/Output)/Outputs/Movi_7 <-> InputData1 (Standard 10 PI)/PI 0001
//     Movi_1 (TC EtherNet/IP Slave)/Assembly 2 (Input/Output)/Outputs/Movi_7 @bit 48 <-> InputData1 (Standard 10 PI)/PI 0004
//     Movi_1 (TC EtherNet/IP Slave)/Assembly 2 (Input/Output)/Outputs/Movi_7 @bit 64 <-> InputData1 (Standard 10 PI)/PI 0005
//     Movi_1 (TC EtherNet/IP Slave)/Assembly 2 (Input/Output)/Outputs/Movi_7 @bit 80 <-> InputData1 (Standard 10 PI)/PI 0006
//     Movi_1 (TC EtherNet/IP Slave)/Assembly 2 (Input/Output)/Outputs/Movi_7 @bit 144 <-> InputData1 (Standard 10 PI)/PI 0010
//   SLOT-00 BACKPLANE (EtherCAT) <-> Field_Network (TC3 EIP Adapter)/BFIO (TC EtherNet/IP Slave)
//     MCP-IOLINK (EP6224-2022)/Module 4 (IO-Link Slave)/IO-Link Port2_out/Port2: process data[0] <-> Assembly 1 (Input/Output)/Inputs/M2S_BFIO_300
//     MCP-IOLINK (EP6224-2022)/Module 4 (IO-Link Slave)/IO-Link Port2_out/Port2: process data[2] <-> Assembly 1 (Input/Output)/Inputs/M2S_BFIO_302
//     MCP-IOLINK (EP6224-2022)/Module 4 (IO-Link Slave)/IO-Link Port2_out/Port2: process data[3] <-> Assembly 1 (Input/Output)/Inputs/M2S_BFIO_303
//     MCP-IOLINK (EP6224-2022)/Module 4 (IO-Link Slave)/IO-Link Port2_out/Port2: process data[4] <-> Assembly 1 (Input/Output)/Inputs/M2S_BFIO_304
//     MCP-IOLINK (EP6224-2022)/Module 4 (IO-Link Slave)/IO-Link Port2_out/Port2: process data[5] <-> Assembly 1 (Input/Output)/Inputs/M2S_BFIO_305
//     MCP-IOLINK (EP6224-2022)/Module 4 (IO-Link Slave)/IO-Link Port2_out/Port2: process data[6] <-> Assembly 1 (Input/Output)/Inputs/M2S_BFIO_306
//     MCP-IOLINK (EP6224-2022)/Module 4 (IO-Link Slave)/IO-Link Port2_out/Port2: process data[7] <-> Assembly 1 (Input/Output)/Inputs/M2S_BFIO_307
//     PWR-Supply (EK1200)/LAS_0600_Slot-01 (EL1018)/Channel 1/Input <-> Assembly 1 (Input/Output)/Outputs/S2M_BFIO_1
//     PWR-Supply (EK1200)/LAS_0600_Slot-02 (EL1018)/Channel 1/Input <-> Assembly 1 (Input/Output)/Outputs/S2M_BFIO_2
//     PWR-Supply (EK1200)/LAS_0600_Slot-01 (EL1018)/Channel 2/Input <-> Assembly 1 (Input/Output)/Outputs/S2M_BFIO_1 @bit 1
//     PWR-Supply (EK1200)/LAS_0600_Slot-01 (EL1018)/Channel 3/Input <-> Assembly 1 (Input/Output)/Outputs/S2M_BFIO_1 @bit 2
//     PWR-Supply (EK1200)/LAS_0600_Slot-01 (EL1018)/Channel 4/Input <-> Assembly 1 (Input/Output)/Outputs/S2M_BFIO_1 @bit 3
//     PWR-Supply (EK1200)/LAS_0600_Slot-01 (EL1018)/Channel 6/Input <-> Assembly 1 (Input/Output)/Outputs/S2M_BFIO_1 @bit 5
//     PWR-Supply (EK1200)/LAS_0600_Slot-01 (EL1018)/Channel 7/Input <-> Assembly 1 (Input/Output)/Outputs/S2M_BFIO_1 @bit 6
//     PWR-Supply (EK1200)/LAS_0600_Slot-01 (EL1018)/Channel 8/Input <-> Assembly 1 (Input/Output)/Outputs/S2M_BFIO_1 @bit 7
//     PWR-Supply (EK1200)/LAS_0600_Slot-02 (EL1018)/Channel 2/Input <-> Assembly 1 (Input/Output)/Outputs/S2M_BFIO_2 @bit 1
//     PWR-Supply (EK1200)/LAS_0600_Slot-02 (EL1018)/Channel 3/Input <-> Assembly 1 (Input/Output)/Outputs/S2M_BFIO_2 @bit 2
//     PWR-Supply (EK1200)/LAS_0600_Slot-02 (EL1018)/Channel 4/Input <-> Assembly 1 (Input/Output)/Outputs/S2M_BFIO_2 @bit 3
//     PWR-Supply (EK1200)/LAS_0600_Slot-02 (EL1018)/Channel 5/Input <-> Assembly 1 (Input/Output)/Outputs/S2M_BFIO_2 @bit 4
//     PWR-Supply (EK1200)/LAS_0600_Slot-02 (EL1018)/Channel 7/Input <-> Assembly 1 (Input/Output)/Outputs/S2M_BFIO_2 @bit 6
//     PWR-Supply (EK1200)/LAS_0600_Slot-02 (EL1018)/Channel 8/Input <-> Assembly 1 (Input/Output)/Outputs/S2M_BFIO_2 @bit 7
//     PWR-Supply (EK1200)/LAS_0600_Slot-05 (EL2008)/Channel 3/Output <-> Assembly 1 (Input/Output)/Inputs/M2S_BFIO_1 @bit 2
//     PWR-Supply (EK1200)/LAS_0600_Slot-05 (EL2008)/Channel 4/Output <-> Assembly 1 (Input/Output)/Inputs/M2S_BFIO_1 @bit 3
//     PWR-Supply (EK1200)/LAS_0600_Slot-05 (EL2008)/Channel 8/Output <-> Assembly 1 (Input/Output)/Inputs/M2S_BFIO_1 @bit 7
//   SLOT-00 BACKPLANE (EtherCAT) <-> Field_Network (TC3 EIP Adapter)/BSIO (TC EtherNet/IP Slave)
//     PWR-Supply (EK1200)/LAS_0600_Slot-04 (EL1904)/Module 1 (FSOES)/TxPDO/FSOE/InputChannel1 <-> Assembly 3 (Input/Output)/Outputs/S2M_BSIO__11
//     PWR-Supply (EK1200)/LAS_0600_Slot-04 (EL1904)/Module 1 (FSOES)/TxPDO/FSOE/InputChannel2 <-> Assembly 3 (Input/Output)/Outputs/S2M_BSIO__11 @bit 1
//     PWR-Supply (EK1200)/LAS_0600_Slot-04 (EL1904)/Module 1 (FSOES)/TxPDO/FSOE/InputChannel3 <-> Assembly 3 (Input/Output)/Outputs/S2M_BSIO__11 @bit 2
//     PWR-Supply (EK1200)/Safety-Ctrl (EL6910)/StandardInputs/Standard Out Var 21 <-> Assembly 3 (Input/Output)/Outputs/S2M_BSIO_1
//     PWR-Supply (EK1200)/Safety-Ctrl (EL6910)/StandardInputs/Standard Out Var 23 <-> Assembly 3 (Input/Output)/Outputs/S2M_BSIO_1 @bit 1
//     PWR-Supply (EK1200)/Safety-Ctrl (EL6910)/StandardInputs/Standard Out Var 24 <-> Assembly 3 (Input/Output)/Outputs/S2M_BSIO_1 @bit 2
//     PWR-Supply (EK1200)/Safety-Ctrl (EL6910)/StandardInputs/Standard Out Var 25 <-> Assembly 3 (Input/Output)/Outputs/S2M_BSIO_1 @bit 3
//     PWR-Supply (EK1200)/Safety-Ctrl (EL6910)/StandardInputs/Standard Out Var 26 <-> Assembly 3 (Input/Output)/Outputs/S2M_BSIO_1 @bit 4
//     PWR-Supply (EK1200)/Safety-Ctrl (EL6910)/StandardInputs/Standard Out Var 28 <-> Assembly 3 (Input/Output)/Outputs/S2M_BSIO_1 @bit 5
//     PWR-Supply (EK1200)/Safety-Ctrl (EL6910)/StandardInputs/Standard Out Var 29 <-> Assembly 3 (Input/Output)/Outputs/S2M_BSIO_1 @bit 6
//     PWR-Supply (EK1200)/Safety-Ctrl (EL6910)/StandardInputs/Standard Out Var 36 <-> Assembly 3 (Input/Output)/Outputs/S2M_BSIO_1 @bit 7
//   SLOT-00 BACKPLANE (EtherCAT) <-> SLOT-00 BACKPLANE (EtherCAT)/PWR-Supply (EK1200)/Safety-Ctrl (EL6910)
//     PWR-Supply (EK1200)/LAS_0600_Slot-04 (EL1904)/Module 1 (FSOES)/RxPDO/FSOE <-> ConnectionInputs/Message_11 TxPDO
//     PWR-Supply (EK1200)/LAS_0600_Slot-04 (EL1904)/Module 1 (FSOES)/TxPDO/FSOE <-> ConnectionOutputs/Message_11 RxPDO
//   SLOT-00 BACKPLANE (EtherCAT) <-> SLOT-04-X600-X601 (EtherCAT)/BSIO-LASB-0622_1 (EP1957-0022)
//     PWR-Supply (EK1200)/Safety-Ctrl (EL6910)/ConnectionInputs/Message_15 TxPDO <-> Module 1 (FSOE)/FSoE Outputs/FSOE
//     PWR-Supply (EK1200)/Safety-Ctrl (EL6910)/ConnectionOutputs/Message_15 RxPDO <-> Module 1 (FSOE)/FSoE Inputs/FSOE
//   SLOT-00 BACKPLANE (EtherCAT) <-> SLOT-04-X600-X601 (EtherCAT)/BSIO-LASB-0623_1 (EP1957-0022)
//     PWR-Supply (EK1200)/Safety-Ctrl (EL6910)/ConnectionOutputs/Message_16 RxPDO <-> Module 1 (FSOE)/FSoE Inputs/FSOE
//   SLOT-00 BACKPLANE (EtherCAT) <-> SLOT-04-X600-X601 (EtherCAT)/BSIO-LASB-0629_1 (EP1957-0022)
//     PWR-Supply (EK1200)/Safety-Ctrl (EL6910)/ConnectionOutputs/Message_18 RxPDO <-> Module 1 (FSOE)/FSoE Inputs/FSOE
//   SLOT-00 BACKPLANE (EtherCAT) <-> SLOT-04-X600-X601 (EtherCAT)/BSIO-LASB-0633_1 (EP1957-0022)
//     PWR-Supply (EK1200)/Safety-Ctrl (EL6910)/ConnectionInputs/Message_17 TxPDO <-> Module 1 (FSOE)/FSoE Outputs/FSOE
//     PWR-Supply (EK1200)/Safety-Ctrl (EL6910)/ConnectionOutputs/Message_17 RxPDO <-> Module 1 (FSOE)/FSoE Inputs/FSOE
//   SLOT-03-X600-X601 (EtherCAT) <-> Field_Network (TC3 EIP Adapter)/BFIO (TC EtherNet/IP Slave)
//     BFIO_LLUB-0635_1 (EP2338-0002)/Channel 14/Output <-> Assembly 1 (Input/Output)/Inputs/M2S_BFIO_11 @bit 5
//     BFIO_LLUB-0635_1 (EP2338-0002)/Channel 1/Input <-> Assembly 1 (Input/Output)/Outputs/S2M_BFIO_13
//     BFIO_LLUB-0635_1 (EP2338-0002)/Channel 2/Input <-> Assembly 1 (Input/Output)/Outputs/S2M_BFIO_13 @bit 1
//     BFIO_LLUB-0635_1 (EP2338-0002)/Channel 3/Input <-> Assembly 1 (Input/Output)/Outputs/S2M_BFIO_13 @bit 2
//     BFIO_LLUB-0635_1 (EP2338-0002)/Channel 4/Input <-> Assembly 1 (Input/Output)/Outputs/S2M_BFIO_13 @bit 3
//     BFIO_LLUB-0635_1 (EP2338-0002)/Channel 5/Input <-> Assembly 1 (Input/Output)/Outputs/S2M_BFIO_13 @bit 4
//     BFIO_LLUB-0635_1 (EP2338-0002)/Channel 6/Input <-> Assembly 1 (Input/Output)/Outputs/S2M_BFIO_13 @bit 5
//     BFIO_LLUB-0635_1 (EP2338-0002)/Channel 7/Input <-> Assembly 1 (Input/Output)/Outputs/S2M_BFIO_13 @bit 6
//     BFIO_LLUB-0635_1 (EP2338-0002)/Channel 8/Input <-> Assembly 1 (Input/Output)/Outputs/S2M_BFIO_13 @bit 7
//     BFIO_LLUB-0635_1 (EP2338-0002)/Channel 9/Output <-> Assembly 1 (Input/Output)/Inputs/M2S_BFIO_11
//     BFIO_LLUB-0636_1(EP2338-0002)/Channel 11/Output <-> Assembly 1 (Input/Output)/Inputs/M2S_BFIO_12 @bit 2
//     BFIO_LLUB-0636_1(EP2338-0002)/Channel 12/Output <-> Assembly 1 (Input/Output)/Inputs/M2S_BFIO_12 @bit 3
//     BFIO_LLUB-0636_1(EP2338-0002)/Channel 16/Output <-> Assembly 1 (Input/Output)/Inputs/M2S_BFIO_12 @bit 7
//     BFIO_LLUB-0636_1(EP2338-0002)/Channel 1/Input <-> Assembly 1 (Input/Output)/Outputs/S2M_BFIO_14
//     BFIO_LLUB-0636_1(EP2338-0002)/Channel 6/Input <-> Assembly 1 (Input/Output)/Outputs/S2M_BFIO_14 @bit 5
//     BSIO_LLUB-0639_2 (EP2338-0002)/Channel 11/Output <-> Assembly 1 (Input/Output)/Inputs/M2S_BFIO_13 @bit 2
//     BSIO_LLUB-0639_2 (EP2338-0002)/Channel 12/Output <-> Assembly 1 (Input/Output)/Inputs/M2S_BFIO_13 @bit 3
//     BSIO_LLUB-0639_2 (EP2338-0002)/Channel 13/Output <-> Assembly 1 (Input/Output)/Inputs/M2S_BFIO_13 @bit 4
//     BSIO_LLUB-0639_2 (EP2338-0002)/Channel 16/Output <-> Assembly 1 (Input/Output)/Inputs/M2S_BFIO_13 @bit 7
//     BSIO_LLUB-0639_2 (EP2338-0002)/Channel 1/Input <-> Assembly 1 (Input/Output)/Outputs/S2M_BFIO_15
//     BSIO_LLUB-0639_2 (EP2338-0002)/Channel 6/Input <-> Assembly 1 (Input/Output)/Outputs/S2M_BFIO_15 @bit 5
//     BSIO_LLUB-0639_2 (EP2338-0002)/Channel 7/Input <-> Assembly 1 (Input/Output)/Outputs/S2M_BFIO_15 @bit 6
//     IOLINK_LLUB-0639_1 (EP6224-2022)/Module 4 (IO-Link Slave)/IO-Link Port2_out/Port2: process data[0] <-> Assembly 1 (Input/Output)/Inputs/M2S_BFIO_300
//     IOLINK_LLUB-0639_1 (EP6224-2022)/Module 4 (IO-Link Slave)/IO-Link Port2_out/Port2: process data[3] <-> Assembly 1 (Input/Output)/Inputs/M2S_BFIO_303
//     IOLINK_LLUB-0639_1 (EP6224-2022)/Module 4 (IO-Link Slave)/IO-Link Port2_out/Port2: process data[4] <-> Assembly 1 (Input/Output)/Inputs/M2S_BFIO_304
//     IOLINK_LLUB-0639_1 (EP6224-2022)/Module 4 (IO-Link Slave)/IO-Link Port2_out/Port2: process data[5] <-> Assembly 1 (Input/Output)/Inputs/M2S_BFIO_305
//     IOLINK_LLUB-0639_1 (EP6224-2022)/Module 4 (IO-Link Slave)/IO-Link Port2_out/Port2: process data[6] <-> Assembly 1 (Input/Output)/Inputs/M2S_BFIO_306
//     LLU-0200 Coupler (EK1100)/LLU_0200_Slot-01 (EL1018)/Channel 3/Input <-> Assembly 1 (Input/Output)/Outputs/S2M_BFIO_10 @bit 2
//     LLU-0200 Coupler (EK1100)/LLU_0200_Slot-01 (EL1018)/Channel 4/Input <-> Assembly 1 (Input/Output)/Outputs/S2M_BFIO_10 @bit 3
//     LLU-0200 Coupler (EK1100)/LLU_0200_Slot-01 (EL1018)/Channel 8/Input <-> Assembly 1 (Input/Output)/Outputs/S2M_BFIO_10 @bit 7
//     LLU-0200 Coupler (EK1100)/LLU_0200_Slot-03 (EL1018)/Channel 2/Input <-> Assembly 1 (Input/Output)/Outputs/S2M_BFIO_12 @bit 1
//     LLU-0200 Coupler (EK1100)/LLU_0200_Slot-03 (EL1018)/Channel 3/Input <-> Assembly 1 (Input/Output)/Outputs/S2M_BFIO_12 @bit 2
//     LLU-0200 Coupler (EK1100)/LLU_0200_Slot-03 (EL1018)/Channel 4/Input <-> Assembly 1 (Input/Output)/Outputs/S2M_BFIO_12 @bit 3
//     LLU-0200 Coupler (EK1100)/LLU_0200_Slot-03 (EL1018)/Channel 6/Input <-> Assembly 1 (Input/Output)/Outputs/S2M_BFIO_12 @bit 5
//     LLU-0200 Coupler (EK1100)/LLU_0200_Slot-03 (EL1018)/Channel 7/Input <-> Assembly 1 (Input/Output)/Outputs/S2M_BFIO_12 @bit 6
//     LLU-0200 Coupler (EK1100)/LLU_0200_Slot-03 (EL1018)/Channel 8/Input <-> Assembly 1 (Input/Output)/Outputs/S2M_BFIO_12 @bit 7
//     LLU-0200 Coupler (EK1100)/LLU_0200_Slot-02(EL1018)/Channel 1/Input <-> Assembly 1 (Input/Output)/Outputs/S2M_BFIO_11
//     LLU-0200 Coupler (EK1100)/LLU_0200_Slot-02(EL1018)/Channel 4/Input <-> Assembly 1 (Input/Output)/Outputs/S2M_BFIO_11 @bit 3
//     LLU-0200 Coupler (EK1100)/LLU_0200_Slot-02(EL1018)/Channel 5/Input <-> Assembly 1 (Input/Output)/Outputs/S2M_BFIO_11 @bit 4
//     LLU-0200 Coupler (EK1100)/LLU_0200_Slot-02(EL1018)/Channel 6/Input <-> Assembly 1 (Input/Output)/Outputs/S2M_BFIO_11 @bit 5
//     LLU-0200 Coupler (EK1100)/LLU_0200_Slot-03 (EL1018)/Channel 1/Input <-> Assembly 1 (Input/Output)/Outputs/S2M_BFIO_12
//     LLU-0200 Coupler (EK1100)/LLU_0200_Slot-05 (EL2008)/Channel 1/Output <-> Assembly 1 (Input/Output)/Inputs/M2S_BFIO_10
//   SLOT-03-X600-X601 (EtherCAT) <-> Field_Network (TC3 EIP Adapter)/BSIO (TC EtherNet/IP Slave)
//     BSIO_LLUB-0635_1 (EP1957-0022)/Module 1 (FSOE)/FSoE Inputs/FSOE/FSIN Module 1.Channel 1.Input <-> Assembly 3 (Input/Output)/Outputs/S2M_BSIO__33
//     BSIO_LLUB-0636_1 (EP1957-0022)/Module 1 (FSOE)/FSoE Inputs/FSOE/FSIN Module 1.Channel 1.Input <-> Assembly 3 (Input/Output)/Outputs/S2M_BSIO__34
//     BSIO_LLUB-0639_2 (EP1957-0022)/Module 1 (FSOE)/FSoE Inputs/FSOE/FSIN Module 1.Channel 1.Input <-> Assembly 3 (Input/Output)/Outputs/S2M_BSIO__36
//     BSIO_LLUB-0635_1 (EP1957-0022)/Module 1 (FSOE)/FSoE Inputs/FSOE/FSIN Module 1.Channel 2.Input <-> Assembly 3 (Input/Output)/Outputs/S2M_BSIO__33 @bit 1
//     BSIO_LLUB-0635_1 (EP1957-0022)/Module 1 (FSOE)/FSoE Inputs/FSOE/FSIN Module 2.Channel 1.Input <-> Assembly 3 (Input/Output)/Outputs/S2M_BSIO__33 @bit 2
//     BSIO_LLUB-0635_1 (EP1957-0022)/Module 1 (FSOE)/FSoE Inputs/FSOE/FSIN Module 2.Channel 2.Input <-> Assembly 3 (Input/Output)/Outputs/S2M_BSIO__33 @bit 3
//     BSIO_LLUB-0635_1 (EP1957-0022)/Module 1 (FSOE)/FSoE Inputs/FSOE/FSIN Module 3.Channel 1.Input <-> Assembly 3 (Input/Output)/Outputs/S2M_BSIO__33 @bit 4
//     BSIO_LLUB-0635_1 (EP1957-0022)/Module 1 (FSOE)/FSoE Inputs/FSOE/FSIN Module 3.Channel 2.Input <-> Assembly 3 (Input/Output)/Outputs/S2M_BSIO__33 @bit 5
//     BSIO_LLUB-0635_1 (EP1957-0022)/Module 1 (FSOE)/FSoE Inputs/FSOE/FSIN Module 4.Channel 1.Input <-> Assembly 3 (Input/Output)/Outputs/S2M_BSIO__33 @bit 6
//     BSIO_LLUB-0639_2 (EP1957-0022)/Module 1 (FSOE)/FSoE Inputs/FSOE/FSIN Module 1.Channel 2.Input <-> Assembly 3 (Input/Output)/Outputs/S2M_BSIO__36 @bit 1
//     BSIO_LLUB-0639_2 (EP1957-0022)/Module 1 (FSOE)/FSoE Inputs/FSOE/FSIN Module 3.Channel 1.Input <-> Assembly 3 (Input/Output)/Outputs/S2M_BSIO__36 @bit 4
//     BSIO_LLUB-0639_2 (EP1957-0022)/Module 1 (FSOE)/FSoE Inputs/FSOE/FSIN Module 3.Channel 2.Input <-> Assembly 3 (Input/Output)/Outputs/S2M_BSIO__36 @bit 5
//     BSIO_LLUB-0639_3 (EP1957-0022)/Module 1 (FSOE)/FSoE Inputs/FSOE/FSIN Module 1.Channel 2.Input <-> Assembly 3 (Input/Output)/Outputs/S2M_BSIO__37 @bit 1
//     BSIO_LLUB-0639_3 (EP1957-0022)/Module 1 (FSOE)/FSoE Inputs/FSOE/FSIN Module 2.Channel 1.Input <-> Assembly 3 (Input/Output)/Outputs/S2M_BSIO__37 @bit 2
//     BSIO_LLUB-0639_3 (EP1957-0022)/Module 1 (FSOE)/FSoE Inputs/FSOE/FSIN Module 3.Channel 1.Input <-> Assembly 3 (Input/Output)/Outputs/S2M_BSIO__37 @bit 4
//     BSIO_LLUB-0639_3 (EP1957-0022)/Module 1 (FSOE)/FSoE Inputs/FSOE/FSIN Module 3.Channel 2.Input <-> Assembly 3 (Input/Output)/Outputs/S2M_BSIO__37 @bit 5
//     BSIO_LLUB-0639_3 (EP1957-0022)/Module 1 (FSOE)/FSoE Inputs/FSOE/FSIN Module 4.Channel 1.Input <-> Assembly 3 (Input/Output)/Outputs/S2M_BSIO__37 @bit 6
//     BSIO_LLUB-0639_1  (EP1957-0022)/Module 1 (FSOE)/FSoE Inputs/FSOE/FSIN Module 1.Channel 1.Input <-> Assembly 3 (Input/Output)/Outputs/S2M_BSIO__35
//     BSIO_LLUB-0639_1  (EP1957-0022)/Module 1 (FSOE)/FSoE Inputs/FSOE/FSIN Module 2.Channel 2.Input <-> Assembly 3 (Input/Output)/Outputs/S2M_BSIO__35 @bit 3
//     BSIO_LLUB-0639_1  (EP1957-0022)/Module 1 (FSOE)/FSoE Inputs/FSOE/FSIN Module 4.Channel 1.Input <-> Assembly 3 (Input/Output)/Outputs/S2M_BSIO__35 @bit 6
//     BSIO_LLUB-0639_1  (EP1957-0022)/Module 1 (FSOE)/FSoE Inputs/FSOE/FSIN Module 4.Channel 2.Input <-> Assembly 3 (Input/Output)/Outputs/S2M_BSIO__35 @bit 7
//     LLU-0200 Coupler (EK1100)/LLU_0200_Slot-04 (EL1904)/Module 1 (FSOES)/TxPDO/FSOE/InputChannel1 <-> Assembly 3 (Input/Output)/Outputs/S2M_BSIO__31
//     LLU-0200 Coupler (EK1100)/LLU_0200_Slot-04 (EL1904)/Module 1 (FSOES)/TxPDO/FSOE/InputChannel2 <-> Assembly 3 (Input/Output)/Outputs/S2M_BSIO__31 @bit 1
//     LLU-0200 Coupler (EK1100)/LLU_0200_Slot-04 (EL1904)/Module 1 (FSOES)/TxPDO/FSOE/InputChannel3 <-> Assembly 3 (Input/Output)/Outputs/S2M_BSIO__31 @bit 2
//   SLOT-03-X600-X601 (EtherCAT) <-> Field_Network (TC3 EIP Adapter)/Movi_1 (TC EtherNet/IP Slave)
//     MOVI_LLUB-0241 (MOVIMOT+MFE72A)/OutputData1 (Standard 10 PO)/PO 0002 <-> Assembly 2 (Input/Output)/Inputs/Movi_14 @bit 16
//     MOVI_LLUB-0241 (MOVIMOT+MFE72A)/OutputData1 (Standard 10 PO)/PO 0007 <-> Assembly 2 (Input/Output)/Inputs/Movi_14 @bit 96
//     MOVI_LLUB-0251 (MOVIMOT+MFE72A)/OutputData1 (Standard 10 PO)/PO 0004 <-> Assembly 2 (Input/Output)/Inputs/Movi_15 @bit 48
//     MOVI_LLUB-0251 (MOVIMOT+MFE72A)/OutputData1 (Standard 10 PO)/PO 0009 <-> Assembly 2 (Input/Output)/Inputs/Movi_15 @bit 128
//     MOVI_LLUB-0251 (MOVIMOT+MFE72A)/OutputData1 (Standard 10 PO)/PO 0010 <-> Assembly 2 (Input/Output)/Inputs/Movi_15 @bit 144
//     MOVI_LLUB-0637 (MOVIMOT+MFE72A)/OutputData1 (Standard 10 PO)/PO 0002 <-> Assembly 2 (Input/Output)/Inputs/Movi_13 @bit 16
//     MOVI_LLUB-0637 (MOVIMOT+MFE72A)/OutputData1 (Standard 10 PO)/PO 0003 <-> Assembly 2 (Input/Output)/Inputs/Movi_13 @bit 32
//     MOVI_LLUB-0637 (MOVIMOT+MFE72A)/OutputData1 (Standard 10 PO)/PO 0004 <-> Assembly 2 (Input/Output)/Inputs/Movi_13 @bit 48
//     MOVI_LLUB-0637 (MOVIMOT+MFE72A)/OutputData1 (Standard 10 PO)/PO 0005 <-> Assembly 2 (Input/Output)/Inputs/Movi_13 @bit 64
//     MOVI_LLUB-0637 (MOVIMOT+MFE72A)/OutputData1 (Standard 10 PO)/PO 0006 <-> Assembly 2 (Input/Output)/Inputs/Movi_13 @bit 80
//     MOVI_LLUB-0637 (MOVIMOT+MFE72A)/OutputData1 (Standard 10 PO)/PO 0007 <-> Assembly 2 (Input/Output)/Inputs/Movi_13 @bit 96
//     MOVI_LLUB-0637 (MOVIMOT+MFE72A)/OutputData1 (Standard 10 PO)/PO 0008 <-> Assembly 2 (Input/Output)/Inputs/Movi_13 @bit 112
//     MOVI_LLUB-0637 (MOVIMOT+MFE72A)/OutputData1 (Standard 10 PO)/PO 0009 <-> Assembly 2 (Input/Output)/Inputs/Movi_13 @bit 128
//     MOVI_LLUB-0637 (MOVIMOT+MFE72A)/OutputData1 (Standard 10 PO)/PO 0010 <-> Assembly 2 (Input/Output)/Inputs/Movi_13 @bit 144
//     MOVI_LLUB-0638 (MOVIMOT+MFE72A)/OutputData1 (Standard 10 PO)/PO 0003 <-> Assembly 2 (Input/Output)/Inputs/Movi_17 @bit 32
//     MOVI_LLUB-0638 (MOVIMOT+MFE72A)/OutputData1 (Standard 10 PO)/PO 0004 <-> Assembly 2 (Input/Output)/Inputs/Movi_17 @bit 48
//     MOVI_LLUB-0638 (MOVIMOT+MFE72A)/OutputData1 (Standard 10 PO)/PO 0005 <-> Assembly 2 (Input/Output)/Inputs/Movi_17 @bit 64
//     MOVI_LLUB-0638 (MOVIMOT+MFE72A)/OutputData1 (Standard 10 PO)/PO 0009 <-> Assembly 2 (Input/Output)/Inputs/Movi_17 @bit 128
//     MOVI_LLUB-0638 (MOVIMOT+MFE72A)/OutputData1 (Standard 10 PO)/PO 0010 <-> Assembly 2 (Input/Output)/Inputs/Movi_17 @bit 144
//     MOVI_LLUB-0635 (MOVITRAC+FSE24B)/OutputData1  (Standard 3 PO)/PO 0002 <-> Assembly 2 (Input/Output)/Inputs/Movi_19 @bit 1
//     MOVI_LLUB-0636 (MOVITRAC+FSE24B)/OutputData1  (Standard 3 PO)/PO 0002 <-> Assembly 2 (Input/Output)/Inputs/Movi_18 @bit 16
//     MOVI_LLUB-0636 (MOVITRAC+FSE24B)/OutputData1  (Standard 3 PO)/PO 0003 <-> Assembly 2 (Input/Output)/Inputs/Movi_18 @bit 32
//     MOVI_LLUB-0637 (MOVIMOT+MFE72A)/OutputData1 (Standard 10 PO)/PO 0001 <-> Assembly 2 (Input/Output)/Inputs/Movi_13
//   SLOT-04-X600-X601 (EtherCAT) <-> Field_Network (TC3 EIP Adapter)/BFIO (TC EtherNet/IP Slave)
//     BFIO-LASB-0620_1 (EP2338-0002)/Channel 10/Output <-> Assembly 1 (Input/Output)/Inputs/M2S_BFIO_3 @bit 1
//     BFIO-LASB-0620_1 (EP2338-0002)/Channel 11/Output <-> Assembly 1 (Input/Output)/Inputs/M2S_BFIO_3 @bit 2
//     BFIO-LASB-0620_1 (EP2338-0002)/Channel 12/Output <-> Assembly 1 (Input/Output)/Inputs/M2S_BFIO_3 @bit 3
//     BFIO-LASB-0620_1 (EP2338-0002)/Channel 13/Output <-> Assembly 1 (Input/Output)/Inputs/M2S_BFIO_3 @bit 4
//     BFIO-LASB-0620_1 (EP2338-0002)/Channel 15/Output <-> Assembly 1 (Input/Output)/Inputs/M2S_BFIO_3 @bit 6
//     BFIO-LASB-0620_1 (EP2338-0002)/Channel 16/Output <-> Assembly 1 (Input/Output)/Inputs/M2S_BFIO_3 @bit 7
//     BFIO-LASB-0622_1 (EP2338-0002)/Channel 10/Output <-> Assembly 1 (Input/Output)/Inputs/M2S_BFIO_2 @bit 1
//     BFIO-LASB-0622_1 (EP2338-0002)/Channel 11/Output <-> Assembly 1 (Input/Output)/Inputs/M2S_BFIO_2 @bit 2
//     BFIO-LASB-0622_1 (EP2338-0002)/Channel 15/Output <-> Assembly 1 (Input/Output)/Inputs/M2S_BFIO_2 @bit 6
//     BFIO-LASB-0622_1 (EP2338-0002)/Channel 16/Output <-> Assembly 1 (Input/Output)/Inputs/M2S_BFIO_2 @bit 7
//     BFIO-LASB-0620_1 (EP2338-0002)/Channel 1/Input <-> Assembly 1 (Input/Output)/Outputs/S2M_BFIO_5
//     BFIO-LASB-0622_1 (EP2338-0002)/Channel 1/Input <-> Assembly 1 (Input/Output)/Outputs/S2M_BFIO_4
//     BFIO-LASB-0620_1 (EP2338-0002)/Channel 2/Input <-> Assembly 1 (Input/Output)/Outputs/S2M_BFIO_5 @bit 1
//     BFIO-LASB-0620_1 (EP2338-0002)/Channel 6/Input <-> Assembly 1 (Input/Output)/Outputs/S2M_BFIO_5 @bit 5
//     BFIO-LASB-0620_1 (EP2338-0002)/Channel 7/Input <-> Assembly 1 (Input/Output)/Outputs/S2M_BFIO_5 @bit 6
//     BFIO-LASB-0620_1 (EP2338-0002)/Channel 8/Input <-> Assembly 1 (Input/Output)/Outputs/S2M_BFIO_5 @bit 7
//     BFIO-LASB-0622_1 (EP2338-0002)/Channel 6/Input <-> Assembly 1 (Input/Output)/Outputs/S2M_BFIO_4 @bit 5
//   SLOT-04-X600-X601 (EtherCAT) <-> Field_Network (TC3 EIP Adapter)/BSIO (TC EtherNet/IP Slave)
//     BSIO-LASB-0622_1 (EP1957-0022)/Module 1 (FSOE)/FSoE Inputs/FSOE/FSIN Module 2.Channel 2.Input <-> Assembly 3 (Input/Output)/Outputs/S2M_BSIO__13 @bit 3
//     BSIO-LASB-0622_1 (EP1957-0022)/Module 1 (FSOE)/FSoE Inputs/FSOE/FSIN Module 4.Channel 1.Input <-> Assembly 3 (Input/Output)/Outputs/S2M_BSIO__13 @bit 6
//     BSIO-LASB-0623_1 (EP1957-0022)/Module 1 (FSOE)/FSoE Inputs/FSOE/FSIN Module 3.Channel 2.Input <-> Assembly 3 (Input/Output)/Outputs/S2M_BSIO__14 @bit 5
//     BSIO-LASB-0625_1 (EP1957-0022)/Module 1 (FSOE)/FSoE Inputs/FSOE/FSIN Module 1.Channel 2.Input <-> Assembly 3 (Input/Output)/Outputs/S2M_BSIO__17 @bit 1
//     BSIO-LASB-0625_1 (EP1957-0022)/Module 1 (FSOE)/FSoE Inputs/FSOE/FSIN Module 2.Channel 1.Input <-> Assembly 3 (Input/Output)/Outputs/S2M_BSIO__17 @bit 2
//     BSIO-LASB-0625_1 (EP1957-0022)/Module 1 (FSOE)/FSoE Inputs/FSOE/FSIN Module 2.Channel 2.Input <-> Assembly 3 (Input/Output)/Outputs/S2M_BSIO__17 @bit 3
//     BSIO-LASB-0625_1 (EP1957-0022)/Module 1 (FSOE)/FSoE Inputs/FSOE/FSIN Module 3.Channel 1.Input <-> Assembly 3 (Input/Output)/Outputs/S2M_BSIO__17 @bit 4
//     BSIO-LASB-0625_1 (EP1957-0022)/Module 1 (FSOE)/FSoE Inputs/FSOE/FSIN Module 3.Channel 2.Input <-> Assembly 3 (Input/Output)/Outputs/S2M_BSIO__17 @bit 5
//     BSIO-LASB-0625_1 (EP1957-0022)/Module 1 (FSOE)/FSoE Inputs/FSOE/FSIN Module 4.Channel 1.Input <-> Assembly 3 (Input/Output)/Outputs/S2M_BSIO__17 @bit 6
//     BSIO-LASB-0625_1 (EP1957-0022)/Module 1 (FSOE)/FSoE Inputs/FSOE/FSIN Module 4.Channel 2.Input <-> Assembly 3 (Input/Output)/Outputs/S2M_BSIO__17 @bit 7
//     BSIO-LASB-0629_1 (EP1957-0022)/Module 1 (FSOE)/FSoE Inputs/FSOE/FSIN Module 1.Channel 2.Input <-> Assembly 3 (Input/Output)/Outputs/S2M_BSIO__16 @bit 1
//     BSIO-LASB-0629_1 (EP1957-0022)/Module 1 (FSOE)/FSoE Inputs/FSOE/FSIN Module 2.Channel 1.Input <-> Assembly 3 (Input/Output)/Outputs/S2M_BSIO__16 @bit 2
//     BSIO-LASB-0629_1 (EP1957-0022)/Module 1 (FSOE)/FSoE Inputs/FSOE/FSIN Module 2.Channel 2.Input <-> Assembly 3 (Input/Output)/Outputs/S2M_BSIO__16 @bit 3
//     BSIO-LASB-0629_1 (EP1957-0022)/Module 1 (FSOE)/FSoE Inputs/FSOE/FSIN Module 3.Channel 1.Input <-> Assembly 3 (Input/Output)/Outputs/S2M_BSIO__16 @bit 4
//     BSIO-LASB-0629_1 (EP1957-0022)/Module 1 (FSOE)/FSoE Inputs/FSOE/FSIN Module 3.Channel 2.Input <-> Assembly 3 (Input/Output)/Outputs/S2M_BSIO__16 @bit 5
//     BSIO-LASB-0629_1 (EP1957-0022)/Module 1 (FSOE)/FSoE Inputs/FSOE/FSIN Module 4.Channel 1.Input <-> Assembly 3 (Input/Output)/Outputs/S2M_BSIO__16 @bit 6
//     BSIO-LASB-0633_1 (EP1957-0022)/Module 1 (FSOE)/FSoE Inputs/FSOE/FSIN Module 1.Channel 2.Input <-> Assembly 3 (Input/Output)/Outputs/S2M_BSIO__15 @bit 1
//     BSIO-LASB-0633_1 (EP1957-0022)/Module 1 (FSOE)/FSoE Inputs/FSOE/FSIN Module 3.Channel 1.Input <-> Assembly 3 (Input/Output)/Outputs/S2M_BSIO__15 @bit 4
//     BSIO-LASB-0633_1 (EP1957-0022)/Module 1 (FSOE)/FSoE Inputs/FSOE/FSIN Module 3.Channel 2.Input <-> Assembly 3 (Input/Output)/Outputs/S2M_BSIO__15 @bit 5
//     BSIO-LASB-0625_1 (EP1957-0022)/Module 1 (FSOE)/FSoE Inputs/FSOE/FSIN Module 1.Channel 1.Input <-> Assembly 3 (Input/Output)/Outputs/S2M_BSIO__17
//     BSIO-LASB-0633_1 (EP1957-0022)/Module 1 (FSOE)/FSoE Inputs/FSOE/FSIN Module 1.Channel 1.Input <-> Assembly 3 (Input/Output)/Outputs/S2M_BSIO__15
//   SLOT-04-X600-X601 (EtherCAT) <-> Field_Network (TC3 EIP Adapter)/Movi_1 (TC EtherNet/IP Slave)
//     MOVI-LASB-0623 (MOVIMOT+MFE72A)/InputData1 (Standard 10 PI)/PI 0002 <-> Assembly 2 (Input/Output)/Outputs/Movi_10 @bit 16
//     MOVI-LASB-0623 (MOVIMOT+MFE72A)/InputData1 (Standard 10 PI)/PI 0003 <-> Assembly 2 (Input/Output)/Outputs/Movi_10 @bit 32
//     MOVI-LASB-0623 (MOVIMOT+MFE72A)/InputData1 (Standard 10 PI)/PI 0004 <-> Assembly 2 (Input/Output)/Outputs/Movi_10 @bit 48
//     MOVI-LASB-0623 (MOVIMOT+MFE72A)/InputData1 (Standard 10 PI)/PI 0005 <-> Assembly 2 (Input/Output)/Outputs/Movi_10 @bit 64
//     MOVI-LASB-0623 (MOVIMOT+MFE72A)/InputData1 (Standard 10 PI)/PI 0007 <-> Assembly 2 (Input/Output)/Outputs/Movi_10 @bit 96
//     MOVI-LASB-0623 (MOVIMOT+MFE72A)/InputData1 (Standard 10 PI)/PI 0008 <-> Assembly 2 (Input/Output)/Outputs/Movi_10 @bit 112
//     MOVI-LASB-0623 (MOVIMOT+MFE72A)/InputData1 (Standard 10 PI)/PI 0009 <-> Assembly 2 (Input/Output)/Outputs/Movi_10 @bit 128
//     MOVI-LASB-0623 (MOVIMOT+MFE72A)/InputData1 (Standard 10 PI)/PI 0010 <-> Assembly 2 (Input/Output)/Outputs/Movi_10 @bit 144
//     MOVI-LASB-0625 (MOVIMOT+MFE72A)/InputData1 (Standard 10 PI)/PI 0002 <-> Assembly 2 (Input/Output)/Outputs/Movi_1 @bit 16
//     MOVI-LASB-0625 (MOVIMOT+MFE72A)/InputData1 (Standard 10 PI)/PI 0003 <-> Assembly 2 (Input/Output)/Outputs/Movi_1 @bit 32
//     MOVI-LASB-0625 (MOVIMOT+MFE72A)/InputData1 (Standard 10 PI)/PI 0004 <-> Assembly 2 (Input/Output)/Outputs/Movi_1 @bit 48
//     MOVI-LASB-0625 (MOVIMOT+MFE72A)/InputData1 (Standard 10 PI)/PI 0005 <-> Assembly 2 (Input/Output)/Outputs/Movi_1 @bit 64
//     MOVI-LASB-0625 (MOVIMOT+MFE72A)/InputData1 (Standard 10 PI)/PI 0007 <-> Assembly 2 (Input/Output)/Outputs/Movi_1 @bit 96
//     MOVI-LASB-0625 (MOVIMOT+MFE72A)/InputData1 (Standard 10 PI)/PI 0008 <-> Assembly 2 (Input/Output)/Outputs/Movi_1 @bit 112
//     MOVI-LASB-0625 (MOVIMOT+MFE72A)/InputData1 (Standard 10 PI)/PI 0009 <-> Assembly 2 (Input/Output)/Outputs/Movi_1 @bit 128
//     MOVI-LASB-0625 (MOVIMOT+MFE72A)/InputData1 (Standard 10 PI)/PI 0010 <-> Assembly 2 (Input/Output)/Outputs/Movi_1 @bit 144
//     MOVI-LASB-0627 (MOVIMOT+MFE72A)/InputData1 (Standard 10 PI)/PI 0005 <-> Assembly 2 (Input/Output)/Outputs/Movi_6 @bit 64
//     MOVI-LASB-0627 (MOVIMOT+MFE72A)/InputData1 (Standard 10 PI)/PI 0006 <-> Assembly 2 (Input/Output)/Outputs/Movi_6 @bit 80
//     MOVI-LASB-0628 (MOVIMOT+MFE72A)/InputData1 (Standard 10 PI)/PI 0002 <-> Assembly 2 (Input/Output)/Outputs/Movi_5 @bit 16
//     MOVI-LASB-0628 (MOVIMOT+MFE72A)/InputData1 (Standard 10 PI)/PI 0007 <-> Assembly 2 (Input/Output)/Outputs/Movi_5 @bit 96
//     MOVI-LASB-0629 (MOVIMOT+MFE72A)/InputData1 (Standard 10 PI)/PI 0009 <-> Assembly 2 (Input/Output)/Outputs/Movi_4 @bit 128
//     MOVI-LASB-0633 (MOVIMOT+MFE72A)/InputData1 (Standard 10 PI)/PI 0002 <-> Assembly 2 (Input/Output)/Outputs/Movi_11 @bit 16
//     MOVI-LASB-0633 (MOVIMOT+MFE72A)/InputData1 (Standard 10 PI)/PI 0003 <-> Assembly 2 (Input/Output)/Outputs/Movi_11 @bit 32
//     MOVI-LASB-0633 (MOVIMOT+MFE72A)/InputData1 (Standard 10 PI)/PI 0004 <-> Assembly 2 (Input/Output)/Outputs/Movi_11 @bit 48
//     MOVI-LASB-0633 (MOVIMOT+MFE72A)/InputData1 (Standard 10 PI)/PI 0005 <-> Assembly 2 (Input/Output)/Outputs/Movi_11 @bit 64
//     MOVI-LASB-0633 (MOVIMOT+MFE72A)/InputData1 (Standard 10 PI)/PI 0006 <-> Assembly 2 (Input/Output)/Outputs/Movi_11 @bit 80
//     MOVI-LASB-0633 (MOVIMOT+MFE72A)/InputData1 (Standard 10 PI)/PI 0007 <-> Assembly 2 (Input/Output)/Outputs/Movi_11 @bit 96
//     MOVI-LASB-0633 (MOVIMOT+MFE72A)/InputData1 (Standard 10 PI)/PI 0008 <-> Assembly 2 (Input/Output)/Outputs/Movi_11 @bit 112
//     MOVI-LASB-0633 (MOVIMOT+MFE72A)/InputData1 (Standard 10 PI)/PI 0009 <-> Assembly 2 (Input/Output)/Outputs/Movi_11 @bit 128
//     MOVI-LASB-0633 (MOVIMOT+MFE72A)/InputData1 (Standard 10 PI)/PI 0010 <-> Assembly 2 (Input/Output)/Outputs/Movi_11 @bit 144
//     MOVI-LASB-0634 (MOVIMOT+MFE72A)/InputData1 (Standard 10 PI)/PI 0003 <-> Assembly 2 (Input/Output)/Outputs/Movi_12 @bit 32
//     MOVI-LASB-0623 (MOVIMOT+MFE72A)/OutputData1 (Standard 10 PO)/PO 0003 <-> Assembly 2 (Input/Output)/Inputs/Movi_10 @bit 32
//     MOVI-LASB-0623 (MOVIMOT+MFE72A)/OutputData1 (Standard 10 PO)/PO 0004 <-> Assembly 2 (Input/Output)/Inputs/Movi_10 @bit 48
//     MOVI-LASB-0623 (MOVIMOT+MFE72A)/OutputData1 (Standard 10 PO)/PO 0005 <-> Assembly 2 (Input/Output)/Inputs/Movi_10 @bit 64
//     MOVI-LASB-0623 (MOVIMOT+MFE72A)/OutputData1 (Standard 10 PO)/PO 0008 <-> Assembly 2 (Input/Output)/Inputs/Movi_10 @bit 112
//     MOVI-LASB-0623 (MOVIMOT+MFE72A)/OutputData1 (Standard 10 PO)/PO 0009 <-> Assembly 2 (Input/Output)/Inputs/Movi_10 @bit 128
//     MOVI-LASB-0623 (MOVIMOT+MFE72A)/OutputData1 (Standard 10 PO)/PO 0010 <-> Assembly 2 (Input/Output)/Inputs/Movi_10 @bit 144
//     MOVI-LASB-0625 (MOVIMOT+MFE72A)/OutputData1 (Standard 10 PO)/PO 0003 <-> Assembly 2 (Input/Output)/Inputs/Movi_1 @bit 32
//     MOVI-LASB-0625 (MOVIMOT+MFE72A)/OutputData1 (Standard 10 PO)/PO 0004 <-> Assembly 2 (Input/Output)/Inputs/Movi_1 @bit 48
//     MOVI-LASB-0625 (MOVIMOT+MFE72A)/OutputData1 (Standard 10 PO)/PO 0005 <-> Assembly 2 (Input/Output)/Inputs/Movi_1 @bit 64
//     MOVI-LASB-0625 (MOVIMOT+MFE72A)/OutputData1 (Standard 10 PO)/PO 0008 <-> Assembly 2 (Input/Output)/Inputs/Movi_1 @bit 112
//     MOVI-LASB-0625 (MOVIMOT+MFE72A)/OutputData1 (Standard 10 PO)/PO 0009 <-> Assembly 2 (Input/Output)/Inputs/Movi_1 @bit 128
//     MOVI-LASB-0625 (MOVIMOT+MFE72A)/OutputData1 (Standard 10 PO)/PO 0010 <-> Assembly 2 (Input/Output)/Inputs/Movi_1 @bit 144
//     MOVI-LASB-0626 (MOVIMOT+MFE72A)/OutputData1 (Standard 10 PO)/PO 0002 <-> Assembly 2 (Input/Output)/Inputs/Movi_3 @bit 16
//     MOVI-LASB-0626 (MOVIMOT+MFE72A)/OutputData1 (Standard 10 PO)/PO 0003 <-> Assembly 2 (Input/Output)/Inputs/Movi_3 @bit 32
//     MOVI-LASB-0626 (MOVIMOT+MFE72A)/OutputData1 (Standard 10 PO)/PO 0004 <-> Assembly 2 (Input/Output)/Inputs/Movi_3 @bit 48
//     MOVI-LASB-0626 (MOVIMOT+MFE72A)/OutputData1 (Standard 10 PO)/PO 0005 <-> Assembly 2 (Input/Output)/Inputs/Movi_3 @bit 64
//     MOVI-LASB-0626 (MOVIMOT+MFE72A)/OutputData1 (Standard 10 PO)/PO 0007 <-> Assembly 2 (Input/Output)/Inputs/Movi_3 @bit 96
//     MOVI-LASB-0626 (MOVIMOT+MFE72A)/OutputData1 (Standard 10 PO)/PO 0008 <-> Assembly 2 (Input/Output)/Inputs/Movi_3 @bit 112
//     MOVI-LASB-0626 (MOVIMOT+MFE72A)/OutputData1 (Standard 10 PO)/PO 0009 <-> Assembly 2 (Input/Output)/Inputs/Movi_3 @bit 128
//     MOVI-LASB-0626 (MOVIMOT+MFE72A)/OutputData1 (Standard 10 PO)/PO 0010 <-> Assembly 2 (Input/Output)/Inputs/Movi_3 @bit 144
//     MOVI-LASB-0627 (MOVIMOT+MFE72A)/OutputData1 (Standard 10 PO)/PO 0007 <-> Assembly 2 (Input/Output)/Inputs/Movi_6 @bit 96
//     MOVI-LASB-0628 (MOVIMOT+MFE72A)/OutputData1 (Standard 10 PO)/PO 0003 <-> Assembly 2 (Input/Output)/Inputs/Movi_5 @bit 32
//     MOVI-LASB-0629 (MOVIMOT+MFE72A)/OutputData1 (Standard 10 PO)/PO 0002 <-> Assembly 2 (Input/Output)/Inputs/Movi_4 @bit 16
//     MOVI-LASB-0629 (MOVIMOT+MFE72A)/OutputData1 (Standard 10 PO)/PO 0003 <-> Assembly 2 (Input/Output)/Inputs/Movi_4 @bit 32
//     MOVI-LASB-0629 (MOVIMOT+MFE72A)/OutputData1 (Standard 10 PO)/PO 0004 <-> Assembly 2 (Input/Output)/Inputs/Movi_4 @bit 48
//     MOVI-LASB-0629 (MOVIMOT+MFE72A)/OutputData1 (Standard 10 PO)/PO 0005 <-> Assembly 2 (Input/Output)/Inputs/Movi_4 @bit 64
//     MOVI-LASB-0629 (MOVIMOT+MFE72A)/OutputData1 (Standard 10 PO)/PO 0006 <-> Assembly 2 (Input/Output)/Inputs/Movi_4 @bit 80
//     MOVI-LASB-0629 (MOVIMOT+MFE72A)/OutputData1 (Standard 10 PO)/PO 0007 <-> Assembly 2 (Input/Output)/Inputs/Movi_4 @bit 96
//     MOVI-LASB-0629 (MOVIMOT+MFE72A)/OutputData1 (Standard 10 PO)/PO 0008 <-> Assembly 2 (Input/Output)/Inputs/Movi_4 @bit 112
//     MOVI-LASB-0629 (MOVIMOT+MFE72A)/OutputData1 (Standard 10 PO)/PO 0009 <-> Assembly 2 (Input/Output)/Inputs/Movi_4 @bit 128
//     MOVI-LASB-0629 (MOVIMOT+MFE72A)/OutputData1 (Standard 10 PO)/PO 0010 <-> Assembly 2 (Input/Output)/Inputs/Movi_4 @bit 144
//     MOVI-LASB-0633 (MOVIMOT+MFE72A)/OutputData1 (Standard 10 PO)/PO 0002 <-> Assembly 2 (Input/Output)/Inputs/Movi_11 @bit 16
//     MOVI-LASB-0633 (MOVIMOT+MFE72A)/OutputData1 (Standard 10 PO)/PO 0003 <-> Assembly 2 (Input/Output)/Inputs/Movi_11 @bit 32
//     MOVI-LASB-0633 (MOVIMOT+MFE72A)/OutputData1 (Standard 10 PO)/PO 0004 <-> Assembly 2 (Input/Output)/Inputs/Movi_11 @bit 48
//     MOVI-LASB-0633 (MOVIMOT+MFE72A)/OutputData1 (Standard 10 PO)/PO 0006 <-> Assembly 2 (Input/Output)/Inputs/Movi_11 @bit 80
//     MOVI-LASB-0633 (MOVIMOT+MFE72A)/OutputData1 (Standard 10 PO)/PO 0007 <-> Assembly 2 (Input/Output)/Inputs/Movi_11 @bit 96
//     MOVI-LASB-0633 (MOVIMOT+MFE72A)/OutputData1 (Standard 10 PO)/PO 0008 <-> Assembly 2 (Input/Output)/Inputs/Movi_11 @bit 112
//     MOVI-LASB-0633 (MOVIMOT+MFE72A)/OutputData1 (Standard 10 PO)/PO 0009 <-> Assembly 2 (Input/Output)/Inputs/Movi_11 @bit 128
//     MOVI-LASB-0634 (MOVIMOT+MFE72A)/OutputData1 (Standard 10 PO)/PO 0002 <-> Assembly 2 (Input/Output)/Inputs/Movi_12 @bit 16
//     MOVI-LASB-0634 (MOVIMOT+MFE72A)/OutputData1 (Standard 10 PO)/PO 0003 <-> Assembly 2 (Input/Output)/Inputs/Movi_12 @bit 32
//     MOVI-LASB-0634 (MOVIMOT+MFE72A)/OutputData1 (Standard 10 PO)/PO 0005 <-> Assembly 2 (Input/Output)/Inputs/Movi_12 @bit 64
//     MOVI-LASB-0634 (MOVIMOT+MFE72A)/OutputData1 (Standard 10 PO)/PO 0006 <-> Assembly 2 (Input/Output)/Inputs/Movi_12 @bit 80
//     MOVI-LASB-0634 (MOVIMOT+MFE72A)/OutputData1 (Standard 10 PO)/PO 0007 <-> Assembly 2 (Input/Output)/Inputs/Movi_12 @bit 96
//     MOVI-LASB-0634 (MOVIMOT+MFE72A)/OutputData1 (Standard 10 PO)/PO 0008 <-> Assembly 2 (Input/Output)/Inputs/Movi_12 @bit 112
//     MOVI-LASB-0634 (MOVIMOT+MFE72A)/OutputData1 (Standard 10 PO)/PO 0010 <-> Assembly 2 (Input/Output)/Inputs/Movi_12 @bit 144
//     MOVI-LASB-0627 (MOVIMOT+MFE72A)/InputData1 (Standard 10 PI)/PI 0001 <-> Assembly 2 (Input/Output)/Outputs/Movi_6
//     MOVI-LASB-0633 (MOVIMOT+MFE72A)/InputData1 (Standard 10 PI)/PI 0001 <-> Assembly 2 (Input/Output)/Outputs/Movi_11
//     MOVI-LASB-0629 (MOVIMOT+MFE72A)/OutputData1 (Standard 10 PO)/PO 0001 <-> Assembly 2 (Input/Output)/Inputs/Movi_4
//     MOVI-LASB-0633 (MOVIMOT+MFE72A)/OutputData1 (Standard 10 PO)/PO 0001 <-> Assembly 2 (Input/Output)/Inputs/Movi_11
//     MOVI-LASB-0634 (MOVIMOT+MFE72A)/OutputData1 (Standard 10 PO)/PO 0001 <-> Assembly 2 (Input/Output)/Inputs/Movi_12
//     MOVI-LASR-0624 (MOVIMOT+MFE72A)/InputData1 (Standard 10 PI)/PI 0001 <-> Assembly 2 (Input/Output)/Outputs/Movi_2
//     MOVI-LASR-0630 (MOVIMOT+MFE72A)/InputData1 (Standard 10 PI)/PI 0001 <-> Assembly 2 (Input/Output)/Outputs/Movi_9
//     MOVI-LASR-0631 (MOVIMOT+MFE72A)/InputData1 (Standard 10 PI)/PI 0001 <-> Assembly 2 (Input/Output)/Outputs/Movi_8
//     MOVI-LASR-0624 (MOVIMOT+MFE72A)/InputData1 (Standard 10 PI)/PI 0002 <-> Assembly 2 (Input/Output)/Outputs/Movi_2 @bit 16
//     MOVI-LASR-0624 (MOVIMOT+MFE72A)/InputData1 (Standard 10 PI)/PI 0003 <-> Assembly 2 (Input/Output)/Outputs/Movi_2 @bit 32
//     MOVI-LASR-0624 (MOVIMOT+MFE72A)/InputData1 (Standard 10 PI)/PI 0004 <-> Assembly 2 (Input/Output)/Outputs/Movi_2 @bit 48
//     MOVI-LASR-0624 (MOVIMOT+MFE72A)/InputData1 (Standard 10 PI)/PI 0005 <-> Assembly 2 (Input/Output)/Outputs/Movi_2 @bit 64
//     MOVI-LASR-0624 (MOVIMOT+MFE72A)/InputData1 (Standard 10 PI)/PI 0006 <-> Assembly 2 (Input/Output)/Outputs/Movi_2 @bit 80
//     MOVI-LASR-0624 (MOVIMOT+MFE72A)/InputData1 (Standard 10 PI)/PI 0007 <-> Assembly 2 (Input/Output)/Outputs/Movi_2 @bit 96
//     MOVI-LASR-0624 (MOVIMOT+MFE72A)/InputData1 (Standard 10 PI)/PI 0008 <-> Assembly 2 (Input/Output)/Outputs/Movi_2 @bit 112
//     MOVI-LASR-0624 (MOVIMOT+MFE72A)/InputData1 (Standard 10 PI)/PI 0009 <-> Assembly 2 (Input/Output)/Outputs/Movi_2 @bit 128
//     MOVI-LASR-0624 (MOVIMOT+MFE72A)/InputData1 (Standard 10 PI)/PI 0010 <-> Assembly 2 (Input/Output)/Outputs/Movi_2 @bit 144
//     MOVI-LASR-0630 (MOVIMOT+MFE72A)/InputData1 (Standard 10 PI)/PI 0004 <-> Assembly 2 (Input/Output)/Outputs/Movi_9 @bit 48
//     MOVI-LASR-0630 (MOVIMOT+MFE72A)/InputData1 (Standard 10 PI)/PI 0005 <-> Assembly 2 (Input/Output)/Outputs/Movi_9 @bit 64
//     MOVI-LASR-0630 (MOVIMOT+MFE72A)/InputData1 (Standard 10 PI)/PI 0006 <-> Assembly 2 (Input/Output)/Outputs/Movi_9 @bit 80
//     MOVI-LASR-0630 (MOVIMOT+MFE72A)/InputData1 (Standard 10 PI)/PI 0009 <-> Assembly 2 (Input/Output)/Outputs/Movi_9 @bit 128
//     MOVI-LASR-0630 (MOVIMOT+MFE72A)/InputData1 (Standard 10 PI)/PI 0010 <-> Assembly 2 (Input/Output)/Outputs/Movi_9 @bit 144
//     MOVI-LASR-0631 (MOVIMOT+MFE72A)/InputData1 (Standard 10 PI)/PI 0002 <-> Assembly 2 (Input/Output)/Outputs/Movi_8 @bit 16
//     MOVI-LASR-0631 (MOVIMOT+MFE72A)/InputData1 (Standard 10 PI)/PI 0005 <-> Assembly 2 (Input/Output)/Outputs/Movi_8 @bit 64
//     MOVI-LASR-0631 (MOVIMOT+MFE72A)/InputData1 (Standard 10 PI)/PI 0006 <-> Assembly 2 (Input/Output)/Outputs/Movi_8 @bit 80
//     MOVI-LASR-0631 (MOVIMOT+MFE72A)/InputData1 (Standard 10 PI)/PI 0007 <-> Assembly 2 (Input/Output)/Outputs/Movi_8 @bit 96
//     MOVI-LASR-0632 (MOVIMOT+MFE72A)/InputData1 (Standard 10 PI)/PI 0002 <-> Assembly 2 (Input/Output)/Outputs/Movi_7 @bit 16
//     MOVI-LASR-0632 (MOVIMOT+MFE72A)/InputData1 (Standard 10 PI)/PI 0003 <-> Assembly 2 (Input/Output)/Outputs/Movi_7 @bit 32
//     MOVI-LASR-0632 (MOVIMOT+MFE72A)/InputData1 (Standard 10 PI)/PI 0007 <-> Assembly 2 (Input/Output)/Outputs/Movi_7 @bit 96
//     MOVI-LASR-0632 (MOVIMOT+MFE72A)/InputData1 (Standard 10 PI)/PI 0008 <-> Assembly 2 (Input/Output)/Outputs/Movi_7 @bit 112
//     MOVI-LASR-0632 (MOVIMOT+MFE72A)/InputData1 (Standard 10 PI)/PI 0009 <-> Assembly 2 (Input/Output)/Outputs/Movi_7 @bit 128
//     MOVI-LASR-0624 (MOVIMOT+MFE72A)/OutputData1 (Standard 10 PO)/PO 0001 <-> Assembly 2 (Input/Output)/Inputs/Movi_2
//     MOVI-LASR-0630 (MOVIMOT+MFE72A)/OutputData1 (Standard 10 PO)/PO 0001 <-> Assembly 2 (Input/Output)/Inputs/Movi_9
//     MOVI-LASR-0631 (MOVIMOT+MFE72A)/OutputData1 (Standard 10 PO)/PO 0001 <-> Assembly 2 (Input/Output)/Inputs/Movi_8
//     MOVI-LASR-0624 (MOVIMOT+MFE72A)/OutputData1 (Standard 10 PO)/PO 0002 <-> Assembly 2 (Input/Output)/Inputs/Movi_2 @bit 16
//     MOVI-LASR-0624 (MOVIMOT+MFE72A)/OutputData1 (Standard 10 PO)/PO 0003 <-> Assembly 2 (Input/Output)/Inputs/Movi_2 @bit 32
//     MOVI-LASR-0624 (MOVIMOT+MFE72A)/OutputData1 (Standard 10 PO)/PO 0004 <-> Assembly 2 (Input/Output)/Inputs/Movi_2 @bit 48
//     MOVI-LASR-0624 (MOVIMOT+MFE72A)/OutputData1 (Standard 10 PO)/PO 0007 <-> Assembly 2 (Input/Output)/Inputs/Movi_2 @bit 96
//     MOVI-LASR-0624 (MOVIMOT+MFE72A)/OutputData1 (Standard 10 PO)/PO 0008 <-> Assembly 2 (Input/Output)/Inputs/Movi_2 @bit 112
//     MOVI-LASR-0624 (MOVIMOT+MFE72A)/OutputData1 (Standard 10 PO)/PO 0009 <-> Assembly 2 (Input/Output)/Inputs/Movi_2 @bit 128
//     MOVI-LASR-0630 (MOVIMOT+MFE72A)/OutputData1 (Standard 10 PO)/PO 0005 <-> Assembly 2 (Input/Output)/Inputs/Movi_9 @bit 64
//     MOVI-LASR-0630 (MOVIMOT+MFE72A)/OutputData1 (Standard 10 PO)/PO 0006 <-> Assembly 2 (Input/Output)/Inputs/Movi_9 @bit 80
//     MOVI-LASR-0630 (MOVIMOT+MFE72A)/OutputData1 (Standard 10 PO)/PO 0007 <-> Assembly 2 (Input/Output)/Inputs/Movi_9 @bit 96
//     MOVI-LASR-0630 (MOVIMOT+MFE72A)/OutputData1 (Standard 10 PO)/PO 0010 <-> Assembly 2 (Input/Output)/Inputs/Movi_9 @bit 144
//     MOVI-LASR-0631 (MOVIMOT+MFE72A)/OutputData1 (Standard 10 PO)/PO 0002 <-> Assembly 2 (Input/Output)/Inputs/Movi_8 @bit 16
//     MOVI-LASR-0631 (MOVIMOT+MFE72A)/OutputData1 (Standard 10 PO)/PO 0003 <-> Assembly 2 (Input/Output)/Inputs/Movi_8 @bit 32
//     MOVI-LASR-0631 (MOVIMOT+MFE72A)/OutputData1 (Standard 10 PO)/PO 0007 <-> Assembly 2 (Input/Output)/Inputs/Movi_8 @bit 96
//     MOVI-LASR-0631 (MOVIMOT+MFE72A)/OutputData1 (Standard 10 PO)/PO 0008 <-> Assembly 2 (Input/Output)/Inputs/Movi_8 @bit 112
//     MOVI-LASR-0632 (MOVIMOT+MFE72A)/OutputData1 (Standard 10 PO)/PO 0003 <-> Assembly 2 (Input/Output)/Inputs/Movi_7 @bit 32
//     MOVI-LASR-0632 (MOVIMOT+MFE72A)/OutputData1 (Standard 10 PO)/PO 0004 <-> Assembly 2 (Input/Output)/Inputs/Movi_7 @bit 48
//     MOVI-LASR-0632 (MOVIMOT+MFE72A)/OutputData1 (Standard 10 PO)/PO 0008 <-> Assembly 2 (Input/Output)/Inputs/Movi_7 @bit 112
//     MOVI-LASR-0632 (MOVIMOT+MFE72A)/OutputData1 (Standard 10 PO)/PO 0009 <-> Assembly 2 (Input/Output)/Inputs/Movi_7 @bit 128
//   SLOT-04-X600-X601 (EtherCAT) <-> SLOT-00 BACKPLANE (EtherCAT)/PWR-Supply (EK1200)/Safety-Ctrl (EL6910)
//     BSIO-LASB-0623_1 (EP1957-0022)/Module 1 (FSOE)/FSoE Outputs/FSOE <-> ConnectionInputs/Message_16 TxPDO
//     BSIO-LASB-0625_1 (EP1957-0022)/Module 1 (FSOE)/FSoE Outputs/FSOE <-> ConnectionInputs/Message_19 TxPDO
//     BSIO-LASB-0629_1 (EP1957-0022)/Module 1 (FSOE)/FSoE Outputs/FSOE <-> ConnectionInputs/Message_18 TxPDO
//     BSIO-LASB-0625_1 (EP1957-0022)/Module 1 (FSOE)/FSoE Inputs/FSOE <-> ConnectionOutputs/Message_19 RxPDO
//   Field_IO/Field_IO Instance <-> Field_Network (TC3 EIP Adapter)/BFIO (TC EtherNet/IP Slave)
//     PlcTask Inputs/MAIN.M2S_Heartbeat <-> Assembly 1 (Input/Output)/Inputs/Heartbeat
//     PlcTask Outputs/MAIN.S2M_Heartbeat <-> Assembly 1 (Input/Output)/Outputs/Heartbeat
//   Field_IO/Field_IO Instance <-> SLOT-01-X600-X601 (EtherCAT)
//     PlcTask Inputs/MAIN.Link_State_Slot_01 <-> Inputs/DevState
//   Field_IO/Field_IO Instance <-> SLOT-02-X600-X601 (EtherCAT)
//     PlcTask Inputs/MAIN.Link_State_Slot_02 <-> Inputs/DevState
//   Field_IO/Field_IO Instance <-> SLOT-03-X600-X601 (EtherCAT)
//     PlcTask Inputs/MAIN.Link_State_Slot_03 <-> Inputs/DevState
//   Field_IO/Field_IO Instance <-> SLOT-04-X600-X601 (EtherCAT)
//     PlcTask Inputs/MAIN.Link_State_Slot_04 <-> Inputs/DevState

CONFIGURATION Field_IO
    RESOURCE PLC ON TwinCAT3
        TASK PlcTask(INTERVAL := T#3ms, PRIORITY := 3);
        PROGRAM MAIN WITH PlcTask : MAIN;
    END_RESOURCE
END_CONFIGURATION

// ---- POUs/MAIN.TcPOU
PROGRAM MAIN

VAR
	// Heartbeat signal to Rockwell PLC (Must Inc Every 100ms)
	S2M_Heartbeat AT %Q* : USINT := 0;	
	// Heartbeat signal from Rockwell PLC (Must Inc Every 100ms)
	M2S_Heartbeat AT %I*: USINT := 0; 
	// Heartbeat Duration (Typically 100ms)
	HB_Dur : TIME := TIME#100MS;
	// Flasher Frequency (Typically 10ms)  This is how fast the system will cycle Flashing Events
	Flasher_Frequency : TIME := TIME#125MS;
	
	System_Flasher : Flasher;
	
	System_Flash : INT := 0;
	
	// Heartbeat Slave 2 Master (Update the Heartbeat counter every Heartbeat Cycle)
	HBCtrS2M :HB_S2M;
	
	// Heartbeat Master 2 Slave Check (Must Change State every 3 Heartbeat Cycles)
	HB_M2S : HB_M2S;	
	Link_State_Slot_01 AT %I*: UINT;
	
	Link_State_Slot_02 AT %I*: UINT;
	Link_State_Slot_03 AT %I*: UINT;
	Link_State_Slot_04 AT %I*: UINT;
	LAS_0600_Run AT %Q* :BOOL := FALSE;
	LLU_0200_Run AT %Q* :BOOL := FALSE;
END_VAR

HBCtrS2M(Dur := HB_Dur, Counter := S2M_Heartbeat);		// Update the Heartbeat counter every time the Heartbeat Duration Elapses
HB_M2S(Dur:= (HB_Dur*3), Counter := M2S_Heartbeat); 	// Check the Heartbeat Status of the Rockwell PLC (Must change states within 3 cycles of the Heartbeat Duration
System_Flasher(Flash_Frequency:= Flasher_Frequency, Flasher := System_Flash);	// Create the System Flasher

LAS_0600_Run := HB_M2S.OK;
LLU_0200_Run := HB_M2S.OK;

END_PROGRAM

// ---- POUs/Flasher.TcPOU
FUNCTION_BLOCK Flasher
VAR_INPUT
	Flash_Frequency : TIME := TIME#10ms;
END_VAR
VAR_OUTPUT
END_VAR
VAR_IN_OUT
	Flasher : INT := 0;
END_VAR
VAR
	// Timer for Flash Function
	Flash_Timer: TON;
END_VAR
VAR // added by the converter: edge detectors and wires of the graphical bodies
    _w1 : BOOL;
END_VAR

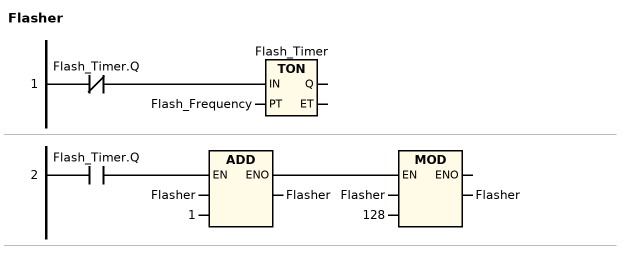
// NETWORK 1
Flash_Timer(IN := NOT Flash_Timer.Q, PT := Flash_Frequency); // TON

// NETWORK 2
_w1 := Flash_Timer.Q;
IF _w1 THEN Flasher := Flasher + 1; END_IF
IF _w1 THEN Flasher := Flasher MOD 128; END_IF

END_FUNCTION_BLOCK

// ---- POUs/HB_S2M.TcPOU
FUNCTION_BLOCK HB_S2M
VAR_INPUT
	Dur : TIME;
END_VAR
VAR_OUTPUT
	ET : TIME;
END_VAR
VAR
	Timer : TON;
END_VAR
VAR_IN_OUT
	Counter : USINT;
END_VAR
VAR // added by the converter: edge detectors and wires of the graphical bodies
    _w1 : BOOL;
END_VAR

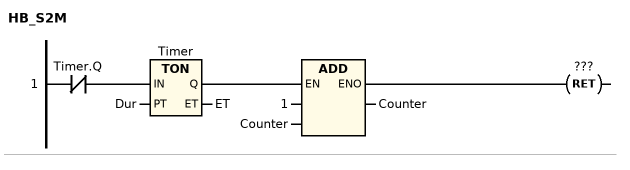
// NETWORK 1
Timer(IN := NOT Timer.Q, PT := Dur, ET => ET); // TON
_w1 := Timer.Q;
IF _w1 THEN Counter := 1 + Counter; END_IF
IF _w1 THEN RETURN; END_IF

END_FUNCTION_BLOCK

// ---- POUs/HB_M2S.TcPOU
FUNCTION_BLOCK HB_M2S
VAR_INPUT
	Dur : TIME;
END_VAR
VAR_OUTPUT
	OK : BOOL;
	ET : TIME;
END_VAR
VAR
	Timer : TON;
	Count_Last : INT;
END_VAR
VAR_IN_OUT
	Counter : USINT;
END_VAR
VAR // added by the converter: edge detectors and wires of the graphical bodies
    _w1, _w2 : BOOL;
END_VAR

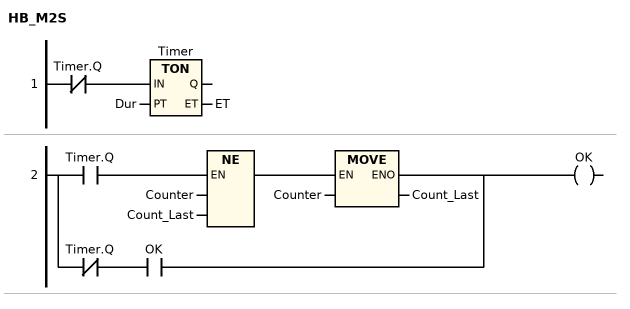
// NETWORK 1
Timer(IN := NOT Timer.Q, PT := Dur, ET => ET); // TON

// NETWORK 2
_w1 := NOT Timer.Q AND OK;
IF NOT _w1 THEN
    _w2 := Timer.Q AND Counter <> Count_Last;
    IF _w2 THEN Count_Last := Counter; END_IF
    _w1 := _w2;
END_IF
OK := _w1;

END_FUNCTION_BLOCK
